LIN {X 0,Y 525.792,Z 279.61,A -85,B 0,C 180,E1 -4784.971,E2 -4784.971} C_VEL
LIN {X 0,Y 524.291,Z 269.507,A -85,B 0,C 180,E1 -4785.168,E2 -4785.168} C_VEL
LIN {X 0,Y 524.691,Z 248.989,A -85,B 0,C 180,E1 -4788.306,E2 -4788.306} C_VEL
LIN {X 0,Y 525.144,Z 230.381,A -85,B 0,C 180,E1 -4791.182,E2 -4791.182} C_VEL
LIN {X 0,Y 525.394,Z 217.304,A -85,B 0,C 180,E1 -4793.241,E2 -4793.241} C_VEL
LIN {X 0,Y 523.911,Z 209.225,A -85,B 0,C 180,E1 -4794.625,E2 -4794.625} C_VEL
LIN {X 0,Y 523.877,Z 209.232,A -85,B 0,C 180,E1 -4797.695,E2 -4797.695} C_VEL
LIN {X 0,Y 523.901,Z 209.222,A -85,B 0,C 180,E1 -4800.844,E2 -4800.844} C_VEL
LIN {X 0,Y 523.896,Z 209.229,A -85,B 0,C 180,E1 -4803.721,E2 -4803.721} C_VEL
LIN {X 0,Y 523.848,Z 209.228,A -85,B 0,C 180,E1 -4806.39,E2 -4806.39} C_VEL
LIN {X 0,Y 523.889,Z 209.223,A -85,B 0,C 180,E1 -4809.086,E2 -4809.086} C_VEL
LIN {X 0,Y 523.876,Z 209.227,A -85,B 0,C 180,E1 -4812.125,E2 -4812.125} C_VEL
LIN {X 0,Y 523.93,Z 209.22,A -85,B 0,C 180,E1 -4815.31,E2 -4815.31} C_VEL
LIN {X 0,Y 523.877,Z 209.223,A -85,B 0,C 180,E1 -4818.698,E2 -4818.698} C_VEL
LIN {X 0,Y 523.884,Z 209.224,A -85,B 0,C 180,E1 -4821.083,E2 -4821.083} C_VEL
LIN {X 0,Y 523.84,Z 209.235,A -85,B 0,C 180,E1 -4823.818,E2 -4823.818} C_VEL
LIN {X 0,Y 523.895,Z 209.221,A -85,B 0,C 180,E1 -4826.629,E2 -4826.629} C_VEL
LIN {X 0,Y 523.907,Z 209.224,A -85,B 0,C 180,E1 -4829.349,E2 -4829.349} C_VEL
LIN {X 0,Y 523.873,Z 209.225,A -85,B 0,C 180,E1 -4832.301,E2 -4832.301} C_VEL
LIN {X 0,Y 523.895,Z 209.227,A -85,B 0,C 180,E1 -4835.423,E2 -4835.423} C_VEL
LIN {X 0,Y 523.934,Z 209.221,A -85,B 0,C 180,E1 -4837.936,E2 -4837.936} C_VEL
LIN {X 0,Y 523.922,Z 209.218,A -85,B 0,C 180,E1 -4840.402,E2 -4840.402} C_VEL
LIN {X 0,Y 523.923,Z 209.218,A -85,B 0,C 180,E1 -4842.832,E2 -4842.832} C_VEL
LIN {X 0,Y 523.957,Z 209.217,A -85,B 0,C 180,E1 -4845.232,E2 -4845.232} C_VEL
LIN {X 0,Y 523.95,Z 209.214,A -85,B 0,C 180,E1 -4848.389,E2 -4848.389} C_VEL
LIN {X 0,Y 523.935,Z 209.225,A -85,B 0,C 180,E1 -4851.511,E2 -4851.511} C_VEL
LIN {X 0,Y 524.022,Z 209.205,A -85,B 0,C 180,E1 -4854.609,E2 -4854.609} C_VEL
LIN {X 0,Y 524.084,Z 209.204,A -85,B 0,C 180,E1 -4857.69,E2 -4857.69} C_VEL
LIN {X 0,Y 524.074,Z 209.201,A -85,B 0,C 180,E1 -4859.996,E2 -4859.996} C_VEL
LIN {X 0,Y 524.016,Z 209.209,A -85,B 0,C 180,E1 -4863.071,E2 -4863.071} C_VEL
LIN {X 0,Y 523.977,Z 209.212,A -85,B 0,C 180,E1 -4866.155,E2 -4866.155} C_VEL
LIN {X 0,Y 523.926,Z 209.223,A -85,B 0,C 180,E1 -4869.258,E2 -4869.258} C_VEL
LIN {X 0,Y 523.973,Z 209.216,A -85,B 0,C 180,E1 -4871.73,E2 -4871.73} C_VEL
LIN {X 0,Y 523.957,Z 209.217,A -85,B 0,C 180,E1 -4875.043,E2 -4875.043} C_VEL
LIN {X 0,Y 523.917,Z 209.22,A -85,B 0,C 180,E1 -4877.965,E2 -4877.965} C_VEL
LIN {X 0,Y 523.928,Z 209.217,A -85,B 0,C 180,E1 -4880.406,E2 -4880.406} C_VEL
LIN {X 0,Y 523.876,Z 209.226,A -85,B 0,C 180,E1 -4882.889,E2 -4882.889} C_VEL
LIN {X 0,Y 523.877,Z 209.232,A -85,B 0,C 180,E1 -4885.416,E2 -4885.416} C_VEL
LIN {X 0,Y 523.92,Z 209.219,A -85,B 0,C 180,E1 -4887.995,E2 -4887.995} C_VEL
LIN {X 0,Y 523.901,Z 209.223,A -85,B 0,C 180,E1 -4890.849,E2 -4890.849} C_VEL
LIN {X 0,Y 523.918,Z 209.222,A -85,B 0,C 180,E1 -4893.73,E2 -4893.73} C_VEL
LIN {X 0,Y 523.859,Z 209.225,A -85,B 0,C 180,E1 -4896.397,E2 -4896.397} C_VEL
LIN {X 0,Y 523.875,Z 209.229,A -85,B 0,C 180,E1 -4899.08,E2 -4899.08} C_VEL
LIN {X 0,Y 523.906,Z 209.22,A -85,B 0,C 180,E1 -4902.115,E2 -4902.115} C_VEL
LIN {X 0,Y 523.905,Z 209.229,A -85,B 0,C 180,E1 -4905.305,E2 -4905.305} C_VEL
LIN {X 0,Y 523.869,Z 209.227,A -85,B 0,C 180,E1 -4906.862,E2 -4906.862} C_VEL
LIN {X 0,Y 523.192,Z 209.315,A -85,B 0,C 180,E1 -4907.504,E2 -4907.504} C_VEL
LIN {X 0,Y 520.325,Z 209.666,A -85,B 0,C 180,E1 -4908.545,E2 -4908.545} C_VEL
LIN {X 0,Y 517.918,Z 209.973,A -85,B 0,C 180,E1 -4909.384,E2 -4909.384} C_VEL
LIN {X 0,Y 516.902,Z 210.093,A -85,B 0,C 180,E1 -4910.032,E2 -4910.032} C_VEL
LIN {X 0,Y 516.828,Z 210.101,A -85,B 0,C 180,E1 -4910.251,E2 -4910.251} C_VEL
LIN {X 0,Y 516.836,Z 210.108,A -85,B 0,C 180,E1 -4913.337,E2 -4913.337} C_VEL
LIN {X 0,Y 516.856,Z 210.098,A -85,B 0,C 180,E1 -4916.118,E2 -4916.118} C_VEL
LIN {X 0,Y 516.835,Z 210.105,A -85,B 0,C 180,E1 -4918.932,E2 -4918.932} C_VEL
LIN {X 0,Y 516.865,Z 210.1,A -85,B 0,C 180,E1 -4921.582,E2 -4921.582} C_VEL
LIN {X 0,Y 516.871,Z 210.096,A -85,B 0,C 180,E1 -4924.208,E2 -4924.208} C_VEL
LIN {X 0,Y 516.842,Z 210.103,A -85,B 0,C 180,E1 -4926.776,E2 -4926.776} C_VEL
LIN {X 0,Y 516.876,Z 210.097,A -85,B 0,C 180,E1 -4929.729,E2 -4929.729} C_VEL
LIN {X 0,Y 516.878,Z 210.097,A -85,B 0,C 180,E1 -4932.595,E2 -4932.595} C_VEL
LIN {X 0,Y 516.875,Z 210.103,A -85,B 0,C 180,E1 -4935.028,E2 -4935.028} C_VEL
LIN {X 0,Y 516.937,Z 210.088,A -85,B 0,C 180,E1 -4938.233,E2 -4938.233} C_VEL
LIN {X 0,Y 516.908,Z 210.096,A -85,B 0,C 180,E1 -4941.399,E2 -4941.399} C_VEL
LIN {X 0,Y 516.956,Z 210.086,A -85,B 0,C 180,E1 -4943.756,E2 -4943.756} C_VEL
LIN {X 0,Y 516.983,Z 210.089,A -85,B 0,C 180,E1 -4946.883,E2 -4946.883} C_VEL
LIN {X 0,Y 517.014,Z 210.078,A -85,B 0,C 180,E1 -4950,E2 -4950} C_VEL
LIN {X 0,Y 516.983,Z 210.09,A -85,B 0,C 180,E1 -4953.117,E2 -4953.117} C_VEL
LIN {X 0,Y 516.956,Z 210.086,A -85,B 0,C 180,E1 -4956.244,E2 -4956.244} C_VEL
LIN {X 0,Y 516.909,Z 210.096,A -85,B 0,C 180,E1 -4958.601,E2 -4958.601} C_VEL
LIN {X 0,Y 516.916,Z 210.095,A -85,B 0,C 180,E1 -4961.825,E2 -4961.825} C_VEL
LIN {X 0,Y 516.944,Z 210.255,A -85,B 0,C 180,E1 -4963.163,E2 -4963.163} C_VEL
LIN {X 0,Y 517.496,Z 216.237,A -85,B 0,C 180,E1 -4964.35,E2 -4964.35} C_VEL
LIN {X 0,Y 517.255,Z 231.009,A -85,B 0,C 180,E1 -4967.188,E2 -4967.188} C_VEL
LIN {X 0,Y 517.241,Z 233.79,A -85,B 0,C 180,E1 -4967.699,E2 -4967.699} C_VEL
LIN {X 0,Y 519.076,Z 243.862,A -85,B 0,C 180,E1 -4967.899,E2 -4967.899} C_VEL
LIN {X 0,Y 518.599,Z 340.175,A -85,B 0,C 180,E1 -4969.262,E2 -4969.262} C_VEL
LIN {X 0,Y 518.408,Z 353.794,A -85,B 0,C 180,E1 -4969.617,E2 -4969.617} C_VEL
LIN {X 0,Y 518.174,Z 366.867,A -85,B 0,C 180,E1 -4970.129,E2 -4970.129} C_VEL
LIN {X 0,Y 517.935,Z 378.637,A -85,B 0,C 180,E1 -4970.762,E2 -4970.762} C_VEL
LIN {X 0,Y 517.624,Z 389.477,A -85,B 0,C 180,E1 -4971.505,E2 -4971.505} C_VEL
LIN {X 0,Y 517.313,Z 399.511,A -85,B 0,C 180,E1 -4972.358,E2 -4972.358} C_VEL
LIN {X 0,Y 516.983,Z 409.671,A -85,B 0,C 180,E1 -4973.43,E2 -4973.43} C_VEL
LIN {X 0,Y 516.771,Z 418.579,A -85,B 0,C 180,E1 -4974.607,E2 -4974.607} C_VEL
LIN {X 0,Y 516.59,Z 425.889,A -85,B 0,C 180,E1 -4975.807,E2 -4975.807} C_VEL
LIN {X 0,Y 516.421,Z 432.17,A -85,B 0,C 180,E1 -4977.122,E2 -4977.122} C_VEL
LIN {X 0,Y 516.366,Z 437.002,A -85,B 0,C 180,E1 -4978.448,E2 -4978.448} C_VEL
LIN {X 0,Y 516.286,Z 439.701,A -85,B 0,C 180,E1 -4979.416,E2 -4979.416} C_VEL
LIN {X 0,Y 516.188,Z 442.581,A -85,B 0,C 180,E1 -4980.949,E2 -4980.949} C_VEL
LIN {X 0,Y 516.18,Z 443.91,A -85,B 0,C 180,E1 -4982.432,E2 -4982.432} C_VEL
LIN {X 0,Y 516.185,Z 443.757,A -85,B 0,C 180,E1 -4983.932,E2 -4983.932} C_VEL
LIN {X 0,Y 516.157,Z 442.467,A -85,B 0,C 180,E1 -4985.231,E2 -4985.231} C_VEL
LIN {X 0,Y 516.309,Z 439.445,A -85,B 0,C 180,E1 -4986.792,E2 -4986.792} C_VEL
LIN {X 0,Y 516.375,Z 434.854,A -85,B 0,C 180,E1 -4988.29,E2 -4988.29} C_VEL
LIN {X 0,Y 516.512,Z 430.235,A -85,B 0,C 180,E1 -4989.417,E2 -4989.417} C_VEL
LIN {X 0,Y 516.652,Z 423.229,A -85,B 0,C 180,E1 -4990.762,E2 -4990.762} C_VEL
LIN {X 0,Y 516.809,Z 416.576,A -85,B 0,C 180,E1 -4991.784,E2 -4991.784} C_VEL
LIN {X 0,Y 517.114,Z 408.481,A -85,B 0,C 180,E1 -4992.806,E2 -4992.806} C_VEL
LIN {X 0,Y 517.385,Z 398.328,A -85,B 0,C 180,E1 -4993.848,E2 -4993.848} C_VEL
LIN {X 0,Y 517.639,Z 388.752,A -85,B 0,C 180,E1 -4994.647,E2 -4994.647} C_VEL
LIN {X 0,Y 517.952,Z 377.818,A -85,B 0,C 180,E1 -4995.385,E2 -4995.385} C_VEL
LIN {X 0,Y 518.222,Z 365.8,A -85,B 0,C 180,E1 -4996.011,E2 -4996.011} C_VEL
LIN {X 0,Y 518.452,Z 352.312,A -85,B 0,C 180,E1 -4996.523,E2 -4996.523} C_VEL
LIN {X 0,Y 518.625,Z 339.718,A -85,B 0,C 180,E1 -4996.837,E2 -4996.837} C_VEL
LIN {X 0,Y 518.974,Z 242.983,A -85,B 0,C 180,E1 -4998.209,E2 -4998.209} C_VEL
LIN {X 0,Y 517.231,Z 233.482,A -85,B 0,C 180,E1 -4998.412,E2 -4998.412} C_VEL
LIN {X 0,Y 517.389,Z 217.337,A -85,B 0,C 180,E1 -5001.338,E2 -5001.338} C_VEL
LIN {X 0,Y 517.232,Z 211.916,A -85,B 0,C 180,E1 -5002.314,E2 -5002.314} C_VEL
LIN {X 0,Y 516.926,Z 210.098,A -85,B 0,C 180,E1 -5002.656,E2 -5002.656} C_VEL
LIN {X 0,Y 516.878,Z 210.098,A -85,B 0,C 180,E1 -5006.037,E2 -5006.037} C_VEL
LIN {X 0,Y 516.856,Z 210.107,A -85,B 0,C 180,E1 -5008.94,E2 -5008.94} C_VEL
LIN {X 0,Y 516.89,Z 210.097,A -85,B 0,C 180,E1 -5011.59,E2 -5011.59} C_VEL
LIN {X 0,Y 516.9,Z 210.093,A -85,B 0,C 180,E1 -5014.216,E2 -5014.216} C_VEL
LIN {X 0,Y 516.841,Z 210.107,A -85,B 0,C 180,E1 -5016.781,E2 -5016.781} C_VEL
LIN {X 0,Y 516.911,Z 210.093,A -85,B 0,C 180,E1 -5019.736,E2 -5019.736} C_VEL
LIN {X 0,Y 516.902,Z 210.098,A -85,B 0,C 180,E1 -5022.601,E2 -5022.601} C_VEL
LIN {X 0,Y 516.917,Z 210.097,A -85,B 0,C 180,E1 -5025.035,E2 -5025.035} C_VEL
LIN {X 0,Y 516.983,Z 210.084,A -85,B 0,C 180,E1 -5028.239,E2 -5028.239} C_VEL
LIN {X 0,Y 516.939,Z 210.089,A -85,B 0,C 180,E1 -5031.404,E2 -5031.404} C_VEL
LIN {X 0,Y 516.979,Z 210.083,A -85,B 0,C 180,E1 -5033.761,E2 -5033.761} C_VEL
LIN {X 0,Y 516.995,Z 210.088,A -85,B 0,C 180,E1 -5036.888,E2 -5036.888} C_VEL
LIN {X 0,Y 517.065,Z 210.073,A -85,B 0,C 180,E1 -5040.004,E2 -5040.004} C_VEL
LIN {X 0,Y 517.062,Z 210.074,A -85,B 0,C 180,E1 -5042.341,E2 -5042.341} C_VEL
LIN {X 0,Y 517.005,Z 210.078,A -85,B 0,C 180,E1 -5045.464,E2 -5045.464} C_VEL
LIN {X 0,Y 516.944,Z 210.087,A -85,B 0,C 180,E1 -5047.818,E2 -5047.818} C_VEL
LIN {X 0,Y 516.935,Z 210.093,A -85,B 0,C 180,E1 -5050.976,E2 -5050.976} C_VEL
LIN {X 0,Y 516.88,Z 210.097,A -85,B 0,C 180,E1 -5054.17,E2 -5054.17} C_VEL
LIN {X 0,Y 516.896,Z 210.102,A -85,B 0,C 180,E1 -5056.594,E2 -5056.594} C_VEL
LIN {X 0,Y 516.888,Z 210.096,A -85,B 0,C 180,E1 -5059.049,E2 -5059.049} C_VEL
LIN {X 0,Y 516.882,Z 210.094,A -85,B 0,C 180,E1 -5061.541,E2 -5061.541} C_VEL
LIN {X 0,Y 516.856,Z 210.104,A -85,B 0,C 180,E1 -5064.354,E2 -5064.354} C_VEL
LIN {X 0,Y 516.874,Z 210.095,A -85,B 0,C 180,E1 -5067.539,E2 -5067.539} C_VEL
LIN {X 0,Y 516.856,Z 210.102,A -85,B 0,C 180,E1 -5070.209,E2 -5070.209} C_VEL
LIN {X 0,Y 516.88,Z 210.096,A -85,B 0,C 180,E1 -5072.951,E2 -5072.951} C_VEL
LIN {X 0,Y 516.816,Z 210.105,A -85,B 0,C 180,E1 -5075.788,E2 -5075.788} C_VEL
LIN {X 0,Y 516.863,Z 210.102,A -85,B 0,C 180,E1 -5078.72,E2 -5078.72} C_VEL
LIN {X 0,Y 516.84,Z 210.103,A -85,B 0,C 180,E1 -5081.785,E2 -5081.785} C_VEL
LIN {X 0,Y 516.901,Z 210.095,A -85,B 0,C 180,E1 -5085.009,E2 -5085.009} C_VEL
LIN {X 0,Y 516.832,Z 210.11,A -85,B 0,C 180,E1 -5088.412,E2 -5088.412} C_VEL
LIN {X 0,Y 516.855,Z 210.099,A -85,B 0,C 180,E1 -5091.283,E2 -5091.283} C_VEL
LIN {X 0,Y 516.831,Z 210.106,A -85,B 0,C 180,E1 -5094.679,E2 -5094.679} C_VEL
LIN {X 0,Y 516.869,Z 210.1,A -85,B 0,C 180,E1 -5097.464,E2 -5097.464} C_VEL
LIN {X 0,Y 516.845,Z 210.108,A -85,B 0,C 180,E1 -5100.492,E2 -5100.492} C_VEL
LIN {X 0,Y 516.818,Z 210.106,A -85,B 0,C 180,E1 -5103.337,E2 -5103.337} C_VEL
LIN {X 0,Y 516.899,Z 210.289,A -85,B 0,C 180,E1 -5105.44,E2 -5105.44} C_VEL
LIN {X 0,Y 518.322,Z 218.758,A -85,B 0,C 180,E1 -5106.846,E2 -5106.846} C_VEL
LIN {X 0,Y 517.95,Z 236.058,A -85,B 0,C 180,E1 -5109.549,E2 -5109.549} C_VEL
LIN {X 0,Y 517.547,Z 254.75,A -85,B 0,C 180,E1 -5112.438,E2 -5112.438} C_VEL
LIN {X 0,Y 517.227,Z 269.021,A -85,B 0,C 180,E1 -5114.622,E2 -5114.622} C_VEL
LIN {X 0,Y 519.018,Z 281.084,A -85,B 0,C 180,E1 -5114.856,E2 -5114.856} C_VEL
LIN {X 0,Y 518.579,Z 377.987,A -85,B 0,C 180,E1 -5116.231,E2 -5116.231} C_VEL
LIN {X 0,Y 518.314,Z 391.113,A -85,B 0,C 180,E1 -5116.574,E2 -5116.574} C_VEL
LIN {X 0,Y 518.039,Z 403.784,A -85,B 0,C 180,E1 -5117.065,E2 -5117.065} C_VEL
LIN {X 0,Y 517.789,Z 415.585,A -85,B 0,C 180,E1 -5117.69,E2 -5117.69} C_VEL
LIN {X 0,Y 517.501,Z 426.729,A -85,B 0,C 180,E1 -5118.445,E2 -5118.445} C_VEL
LIN {X 0,Y 517.219,Z 437.236,A -85,B 0,C 180,E1 -5119.331,E2 -5119.331} C_VEL
LIN {X 0,Y 516.924,Z 445.825,A -85,B 0,C 180,E1 -5120.216,E2 -5120.216} C_VEL
LIN {X 0,Y 516.705,Z 453.75,A -85,B 0,C 180,E1 -5121.198,E2 -5121.198} C_VEL
LIN {X 0,Y 516.529,Z 461.492,A -85,B 0,C 180,E1 -5122.377,E2 -5122.377} C_VEL
LIN {X 0,Y 516.385,Z 468.624,A -85,B 0,C 180,E1 -5123.749,E2 -5123.749} C_VEL
LIN {X 0,Y 516.313,Z 473.37,A -85,B 0,C 180,E1 -5124.924,E2 -5124.924} C_VEL
LIN {X 0,Y 516.354,Z 477,A -85,B 0,C 180,E1 -5126.098,E2 -5126.098} C_VEL
LIN {X 0,Y 516.284,Z 478.87,A -85,B 0,C 180,E1 -5126.879,E2 -5126.879} C_VEL
LIN {X 0,Y 516.263,Z 480.273,A -85,B 0,C 180,E1 -5127.66,E2 -5127.66} C_VEL
LIN {X 0,Y 516.164,Z 481.885,A -85,B 0,C 180,E1 -5129.22,E2 -5129.22} C_VEL
LIN {X 0,Y 516.161,Z 482.105,A -85,B 0,C 180,E1 -5130,E2 -5130} C_VEL
LIN {X 0,Y 516.193,Z 481.283,A -85,B 0,C 180,E1 -5131.56,E2 -5131.56} C_VEL
LIN {X 0,Y 516.263,Z 480.29,A -85,B 0,C 180,E1 -5132.341,E2 -5132.341} C_VEL
LIN {X 0,Y 516.284,Z 478.892,A -85,B 0,C 180,E1 -5133.121,E2 -5133.121} C_VEL
LIN {X 0,Y 516.312,Z 475.95,A -85,B 0,C 180,E1 -5134.293,E2 -5134.293} C_VEL
LIN {X 0,Y 516.369,Z 471.966,A -85,B 0,C 180,E1 -5135.467,E2 -5135.467} C_VEL
LIN {X 0,Y 516.394,Z 466.783,A -85,B 0,C 180,E1 -5136.654,E2 -5136.654} C_VEL
LIN {X 0,Y 516.546,Z 460.374,A -85,B 0,C 180,E1 -5137.82,E2 -5137.82} C_VEL
LIN {X 0,Y 516.758,Z 452.318,A -85,B 0,C 180,E1 -5138.998,E2 -5138.998} C_VEL
LIN {X 0,Y 516.95,Z 444.106,A -85,B 0,C 180,E1 -5139.982,E2 -5139.982} C_VEL
LIN {X 0,Y 517.288,Z 434.094,A -85,B 0,C 180,E1 -5140.965,E2 -5140.965} C_VEL
LIN {X 0,Y 517.569,Z 424.203,A -85,B 0,C 180,E1 -5141.752,E2 -5141.752} C_VEL
LIN {X 0,Y 517.851,Z 413.036,A -85,B 0,C 180,E1 -5142.465,E2 -5142.465} C_VEL
LIN {X 0,Y 518.115,Z 400.511,A -85,B 0,C 180,E1 -5143.082,E2 -5143.082} C_VEL
LIN {X 0,Y 518.395,Z 388.177,A -85,B 0,C 180,E1 -5143.524,E2 -5143.524} C_VEL
LIN {X 0,Y 518.626,Z 375.486,A -85,B 0,C 180,E1 -5143.818,E2 -5143.818} C_VEL
LIN {X 0,Y 518.866,Z 279.935,A -85,B 0,C 180,E1 -5145.168,E2 -5145.168} C_VEL
LIN {X 0,Y 517.279,Z 269.248,A -85,B 0,C 180,E1 -5145.38,E2 -5145.38} C_VEL
LIN {X 0,Y 517.743,Z 248.473,A -85,B 0,C 180,E1 -5148.602,E2 -5148.602} C_VEL
LIN {X 0,Y 518.21,Z 230.161,A -85,B 0,C 180,E1 -5151.479,E2 -5151.479} C_VEL
LIN {X 0,Y 518.434,Z 218.384,A -85,B 0,C 180,E1 -5153.36,E2 -5153.36} C_VEL
LIN {X 0,Y 516.888,Z 210.1,A -85,B 0,C 180,E1 -5154.78,E2 -5154.78} C_VEL
LIN {X 0,Y 516.826,Z 210.11,A -85,B 0,C 180,E1 -5157.881,E2 -5157.881} C_VEL
LIN {X 0,Y 516.842,Z 210.105,A -85,B 0,C 180,E1 -5160.206,E2 -5160.206} C_VEL
LIN {X 0,Y 516.818,Z 210.103,A -85,B 0,C 180,E1 -5162.952,E2 -5162.952} C_VEL
LIN {X 0,Y 516.8,Z 210.114,A -85,B 0,C 180,E1 -5165.785,E2 -5165.785} C_VEL
LIN {X 0,Y 516.853,Z 210.098,A -85,B 0,C 180,E1 -5168.717,E2 -5168.717} C_VEL
LIN {X 0,Y 516.827,Z 210.111,A -85,B 0,C 180,E1 -5171.782,E2 -5171.782} C_VEL
LIN {X 0,Y 516.867,Z 210.097,A -85,B 0,C 180,E1 -5175.001,E2 -5175.001} C_VEL
LIN {X 0,Y 516.832,Z 210.103,A -85,B 0,C 180,E1 -5178.214,E2 -5178.214} C_VEL
LIN {X 0,Y 516.848,Z 210.102,A -85,B 0,C 180,E1 -5181.278,E2 -5181.278} C_VEL
LIN {X 0,Y 516.822,Z 210.102,A -85,B 0,C 180,E1 -5184.675,E2 -5184.675} C_VEL
LIN {X 0,Y 516.864,Z 210.103,A -85,B 0,C 180,E1 -5187.46,E2 -5187.46} C_VEL
LIN {X 0,Y 516.839,Z 210.1,A -85,B 0,C 180,E1 -5190.488,E2 -5190.488} C_VEL
LIN {X 0,Y 516.818,Z 210.107,A -85,B 0,C 180,E1 -5193.333,E2 -5193.333} C_VEL
LIN {X 0,Y 516.868,Z 210.101,A -85,B 0,C 180,E1 -5195.923,E2 -5195.923} C_VEL
LIN {X 0,Y 516.859,Z 210.098,A -85,B 0,C 180,E1 -5198.458,E2 -5198.458} C_VEL
LIN {X 0,Y 516.86,Z 210.098,A -85,B 0,C 180,E1 -5200.95,E2 -5200.95} C_VEL
LIN {X 0,Y 516.867,Z 210.103,A -85,B 0,C 180,E1 -5203.405,E2 -5203.405} C_VEL
LIN {X 0,Y 516.865,Z 210.102,A -85,B 0,C 180,E1 -5205.829,E2 -5205.829} C_VEL
LIN {X 0,Y 516.914,Z 210.092,A -85,B 0,C 180,E1 -5208.229,E2 -5208.229} C_VEL
LIN {X 0,Y 516.908,Z 210.098,A -85,B 0,C 180,E1 -5211.395,E2 -5211.395} C_VEL
LIN {X 0,Y 516.973,Z 210.083,A -85,B 0,C 180,E1 -5214.535,E2 -5214.535} C_VEL
LIN {X 0,Y 517.055,Z 210.08,A -85,B 0,C 180,E1 -5217.659,E2 -5217.659} C_VEL
LIN {X 0,Y 517.044,Z 210.077,A -85,B 0,C 180,E1 -5219.996,E2 -5219.996} C_VEL
LIN {X 0,Y 517.055,Z 210.073,A -85,B 0,C 180,E1 -5222.332,E2 -5222.332} C_VEL
LIN {X 0,Y 516.961,Z 210.094,A -85,B 0,C 180,E1 -5225.456,E2 -5225.456} C_VEL
LIN {X 0,Y 516.907,Z 210.092,A -85,B 0,C 180,E1 -5228.596,E2 -5228.596} C_VEL
LIN {X 0,Y 516.931,Z 210.092,A -85,B 0,C 180,E1 -5231.802,E2 -5231.802} C_VEL
LIN {X 0,Y 516.91,Z 210.096,A -85,B 0,C 180,E1 -5235.137,E2 -5235.137} C_VEL
LIN {X 0,Y 516.885,Z 210.095,A -85,B 0,C 180,E1 -5238.218,E2 -5238.218} C_VEL
LIN {X 0,Y 516.875,Z 210.096,A -85,B 0,C 180,E1 -5240.697,E2 -5240.697} C_VEL
LIN {X 0,Y 516.852,Z 210.099,A -85,B 0,C 180,E1 -5244.069,E2 -5244.069} C_VEL
LIN {X 0,Y 516.871,Z 210.097,A -85,B 0,C 180,E1 -5246.654,E2 -5246.654} C_VEL
LIN {X 0,Y 516.871,Z 210.103,A -85,B 0,C 180,E1 -5249.518,E2 -5249.518} C_VEL
LIN {X 0,Y 516.856,Z 210.098,A -85,B 0,C 180,E1 -5252.539,E2 -5252.539} C_VEL
LIN {X 0,Y 516.824,Z 210.111,A -85,B 0,C 180,E1 -5255.325,E2 -5255.325} C_VEL
LIN {X 0,Y 516.835,Z 210.102,A -85,B 0,C 180,E1 -5257.938,E2 -5257.938} C_VEL
LIN {X 0,Y 516.838,Z 210.102,A -85,B 0,C 180,E1 -5260.737,E2 -5260.737} C_VEL
LIN {X 0,Y 516.837,Z 210.103,A -85,B 0,C 180,E1 -5262.827,E2 -5262.827} C_VEL
LIN {X 0,Y 516.873,Z 210.101,A -85,B 0,C 180,E1 -5265.006,E2 -5265.006} C_VEL
LIN {X 0,Y 516.87,Z 210.096,A -85,B 0,C 180,E1 -5268.394,E2 -5268.394} C_VEL
LIN {X 0,Y 516.828,Z 210.101,A -85,B 0,C 180,E1 -5270.251,E2 -5270.251} C_VEL
LIN {X 0,Y 516.188,Z 210.187,A -85,B 0,C 180,E1 -5270.901,E2 -5270.901} C_VEL
LIN {X 0,Y 513.348,Z 210.542,A -85,B 0,C 180,E1 -5271.957,E2 -5271.957} C_VEL
LIN {X 0,Y 510.926,Z 210.844,A -85,B 0,C 180,E1 -5272.807,E2 -5272.807} C_VEL
LIN {X 0,Y 509.874,Z 210.974,A -85,B 0,C 180,E1 -5273.463,E2 -5273.463} C_VEL
LIN {X 0,Y 509.784,Z 210.982,A -85,B 0,C 180,E1 -5273.686,E2 -5273.686} C_VEL
LIN {X 0,Y 509.805,Z 210.977,A -85,B 0,C 180,E1 -5276.536,E2 -5276.536} C_VEL
LIN {X 0,Y 509.792,Z 210.985,A -85,B 0,C 180,E1 -5279.332,E2 -5279.332} C_VEL
LIN {X 0,Y 509.836,Z 210.972,A -85,B 0,C 180,E1 -5282.052,E2 -5282.052} C_VEL
LIN {X 0,Y 509.821,Z 210.977,A -85,B 0,C 180,E1 -5284.702,E2 -5284.702} C_VEL
LIN {X 0,Y 509.821,Z 210.979,A -85,B 0,C 180,E1 -5287.44,E2 -5287.44} C_VEL
LIN {X 0,Y 509.854,Z 210.971,A -85,B 0,C 180,E1 -5289.843,E2 -5289.843} C_VEL
LIN {X 0,Y 509.843,Z 210.972,A -85,B 0,C 180,E1 -5292.347,E2 -5292.347} C_VEL
LIN {X 0,Y 509.8,Z 210.979,A -85,B 0,C 180,E1 -5295.633,E2 -5295.633} C_VEL
LIN {X 0,Y 509.87,Z 210.974,A -85,B 0,C 180,E1 -5298.874,E2 -5298.874} C_VEL
LIN {X 0,Y 509.904,Z 210.964,A -85,B 0,C 180,E1 -5302.078,E2 -5302.078} C_VEL
LIN {X 0,Y 509.948,Z 210.96,A -85,B 0,C 180,E1 -5304.464,E2 -5304.464} C_VEL
LIN {X 0,Y 509.99,Z 210.955,A -85,B 0,C 180,E1 -5307.631,E2 -5307.631} C_VEL
LIN {X 0,Y 509.985,Z 210.954,A -85,B 0,C 180,E1 -5310,E2 -5310} C_VEL
LIN {X 0,Y 509.924,Z 210.968,A -85,B 0,C 180,E1 -5313.16,E2 -5313.16} C_VEL
LIN {X 0,Y 509.927,Z 210.962,A -85,B 0,C 180,E1 -5316.33,E2 -5316.33} C_VEL
LIN {X 0,Y 509.884,Z 210.973,A -85,B 0,C 180,E1 -5318.72,E2 -5318.72} C_VEL
LIN {X 0,Y 509.885,Z 210.971,A -85,B 0,C 180,E1 -5321.932,E2 -5321.932} C_VEL
LIN {X 0,Y 509.89,Z 211.067,A -85,B 0,C 180,E1 -5323.018,E2 -5323.018} C_VEL
LIN {X 0,Y 510.539,Z 217.685,A -85,B 0,C 180,E1 -5324.346,E2 -5324.346} C_VEL
LIN {X 0,Y 510.238,Z 232.559,A -85,B 0,C 180,E1 -5327.225,E2 -5327.225} C_VEL
LIN {X 0,Y 510.261,Z 233.996,A -85,B 0,C 180,E1 -5327.483,E2 -5327.483} C_VEL
LIN {X 0,Y 512.257,Z 245.073,A -85,B 0,C 180,E1 -5327.706,E2 -5327.706} C_VEL
LIN {X 0,Y 511.722,Z 340.827,A -85,B 0,C 180,E1 -5329.085,E2 -5329.085} C_VEL
LIN {X 0,Y 511.511,Z 354.047,A -85,B 0,C 180,E1 -5329.436,E2 -5329.436} C_VEL
LIN {X 0,Y 511.277,Z 366.832,A -85,B 0,C 180,E1 -5329.942,E2 -5329.942} C_VEL
LIN {X 0,Y 510.998,Z 379.302,A -85,B 0,C 180,E1 -5330.622,E2 -5330.622} C_VEL
LIN {X 0,Y 510.644,Z 390.267,A -85,B 0,C 180,E1 -5331.39,E2 -5331.39} C_VEL
LIN {X 0,Y 510.298,Z 401.247,A -85,B 0,C 180,E1 -5332.355,E2 -5332.355} C_VEL
LIN {X 0,Y 509.972,Z 410.265,A -85,B 0,C 180,E1 -5333.341,E2 -5333.341} C_VEL
LIN {X 0,Y 509.748,Z 419.017,A -85,B 0,C 180,E1 -5334.519,E2 -5334.519} C_VEL
LIN {X 0,Y 509.525,Z 426.382,A -85,B 0,C 180,E1 -5335.752,E2 -5335.752} C_VEL
LIN {X 0,Y 509.354,Z 432.603,A -85,B 0,C 180,E1 -5337.085,E2 -5337.085} C_VEL
LIN {X 0,Y 509.301,Z 437.395,A -85,B 0,C 180,E1 -5338.428,E2 -5338.428} C_VEL
LIN {X 0,Y 509.16,Z 440.923,A -85,B 0,C 180,E1 -5339.795,E2 -5339.795} C_VEL
LIN {X 0,Y 509.094,Z 443.162,A -85,B 0,C 180,E1 -5341.155,E2 -5341.155} C_VEL
LIN {X 0,Y 509.077,Z 444.22,A -85,B 0,C 180,E1 -5342.648,E2 -5342.648} C_VEL
LIN {X 0,Y 509.082,Z 443.935,A -85,B 0,C 180,E1 -5344.087,E2 -5344.087} C_VEL
LIN {X 0,Y 509.104,Z 442.425,A -85,B 0,C 180,E1 -5345.477,E2 -5345.477} C_VEL
LIN {X 0,Y 509.243,Z 439.719,A -85,B 0,C 180,E1 -5346.839,E2 -5346.839} C_VEL
LIN {X 0,Y 509.29,Z 435.891,A -85,B 0,C 180,E1 -5348.145,E2 -5348.145} C_VEL
LIN {X 0,Y 509.432,Z 430.849,A -85,B 0,C 180,E1 -5349.427,E2 -5349.427} C_VEL
LIN {X 0,Y 509.613,Z 423.769,A -85,B 0,C 180,E1 -5350.819,E2 -5350.819} C_VEL
LIN {X 0,Y 509.782,Z 416.879,A -85,B 0,C 180,E1 -5351.898,E2 -5351.898} C_VEL
LIN {X 0,Y 510.106,Z 408.598,A -85,B 0,C 180,E1 -5352.956,E2 -5352.956} C_VEL
LIN {X 0,Y 510.379,Z 399.397,A -85,B 0,C 180,E1 -5353.92,E2 -5353.92} C_VEL
LIN {X 0,Y 510.688,Z 388.417,A -85,B 0,C 180,E1 -5354.852,E2 -5354.852} C_VEL
LIN {X 0,Y 511.027,Z 378.028,A -85,B 0,C 180,E1 -5355.555,E2 -5355.555} C_VEL
LIN {X 0,Y 511.302,Z 366.059,A -85,B 0,C 180,E1 -5356.187,E2 -5356.187} C_VEL
LIN {X 0,Y 511.553,Z 352.701,A -85,B 0,C 180,E1 -5356.702,E2 -5356.702} C_VEL
LIN {X 0,Y 511.738,Z 339.562,A -85,B 0,C 180,E1 -5357.031,E2 -5357.031} C_VEL
LIN {X 0,Y 512.198,Z 244.126,A -85,B 0,C 180,E1 -5358.402,E2 -5358.402} C_VEL
LIN {X 0,Y 510.232,Z 233.768,A -85,B 0,C 180,E1 -5358.621,E2 -5358.621} C_VEL
LIN {X 0,Y 510.416,Z 218.102,A -85,B 0,C 180,E1 -5361.469,E2 -5361.469} C_VEL
LIN {X 0,Y 510.179,Z 212.733,A -85,B 0,C 180,E1 -5362.45,E2 -5362.45} C_VEL
LIN {X 0,Y 509.871,Z 210.977,A -85,B 0,C 180,E1 -5362.792,E2 -5362.792} C_VEL
LIN {X 0,Y 509.825,Z 210.978,A -85,B 0,C 180,E1 -5365.8,E2 -5365.8} C_VEL
LIN {X 0,Y 509.811,Z 210.983,A -85,B 0,C 180,E1 -5368.724,E2 -5368.724} C_VEL
LIN {X 0,Y 509.85,Z 210.979,A -85,B 0,C 180,E1 -5371.161,E2 -5371.161} C_VEL
LIN {X 0,Y 509.877,Z 210.968,A -85,B 0,C 180,E1 -5373.834,E2 -5373.834} C_VEL
LIN {X 0,Y 509.805,Z 210.979,A -85,B 0,C 180,E1 -5376.442,E2 -5376.442} C_VEL
LIN {X 0,Y 509.888,Z 210.967,A -85,B 0,C 180,E1 -5379.85,E2 -5379.85} C_VEL
LIN {X 0,Y 509.858,Z 210.977,A -85,B 0,C 180,E1 -5383.18,E2 -5383.18} C_VEL
LIN {X 0,Y 509.839,Z 210.973,A -85,B 0,C 180,E1 -5385.639,E2 -5385.639} C_VEL
LIN {X 0,Y 509.909,Z 210.971,A -85,B 0,C 180,E1 -5388.88,E2 -5388.88} C_VEL
LIN {X 0,Y 509.903,Z 210.964,A -85,B 0,C 180,E1 -5392.083,E2 -5392.083} C_VEL
LIN {X 0,Y 509.956,Z 210.962,A -85,B 0,C 180,E1 -5394.469,E2 -5394.469} C_VEL
LIN {X 0,Y 510.034,Z 210.947,A -85,B 0,C 180,E1 -5397.635,E2 -5397.635} C_VEL
LIN {X 0,Y 510.051,Z 210.953,A -85,B 0,C 180,E1 -5400.794,E2 -5400.794} C_VEL
LIN {X 0,Y 509.904,Z 210.967,A -85,B 0,C 180,E1 -5403.165,E2 -5403.165} C_VEL
LIN {X 0,Y 509.928,Z 210.963,A -85,B 0,C 180,E1 -5406.334,E2 -5406.334} C_VEL
LIN {X 0,Y 509.875,Z 210.974,A -85,B 0,C 180,E1 -5408.725,E2 -5408.725} C_VEL
LIN {X 0,Y 509.898,Z 210.966,A -85,B 0,C 180,E1 -5411.936,E2 -5411.936} C_VEL
LIN {X 0,Y 509.891,Z 210.967,A -85,B 0,C 180,E1 -5415.246,E2 -5415.246} C_VEL
LIN {X 0,Y 509.853,Z 210.976,A -85,B 0,C 180,E1 -5418.488,E2 -5418.488} C_VEL
LIN {X 0,Y 509.847,Z 210.974,A -85,B 0,C 180,E1 -5421.005,E2 -5421.005} C_VEL
LIN {X 0,Y 509.81,Z 210.975,A -85,B 0,C 180,E1 -5423.568,E2 -5423.568} C_VEL
LIN {X 0,Y 509.799,Z 210.983,A -85,B 0,C 180,E1 -5426.356,E2 -5426.356} C_VEL
LIN {X 0,Y 509.849,Z 210.974,A -85,B 0,C 180,E1 -5428.849,E2 -5428.849} C_VEL
LIN {X 0,Y 509.811,Z 210.976,A -85,B 0,C 180,E1 -5431.594,E2 -5431.594} C_VEL
LIN {X 0,Y 509.834,Z 210.98,A -85,B 0,C 180,E1 -5434.418,E2 -5434.418} C_VEL
LIN {X 0,Y 509.778,Z 210.98,A -85,B 0,C 180,E1 -5437.347,E2 -5437.347} C_VEL
LIN {X 0,Y 509.794,Z 210.986,A -85,B 0,C 180,E1 -5440.389,E2 -5440.389} C_VEL
LIN {X 0,Y 509.796,Z 210.98,A -85,B 0,C 180,E1 -5443.577,E2 -5443.577} C_VEL
LIN {X 0,Y 509.795,Z 210.987,A -85,B 0,C 180,E1 -5446.427,E2 -5446.427} C_VEL
LIN {X 0,Y 509.79,Z 210.98,A -85,B 0,C 180,E1 -5449.614,E2 -5449.614} C_VEL
LIN {X 0,Y 509.763,Z 210.987,A -85,B 0,C 180,E1 -5452.656,E2 -5452.656} C_VEL
LIN {X 0,Y 509.834,Z 210.977,A -85,B 0,C 180,E1 -5455.804,E2 -5455.804} C_VEL
LIN {X 0,Y 509.821,Z 210.981,A -85,B 0,C 180,E1 -5458.728,E2 -5458.728} C_VEL
LIN {X 0,Y 509.798,Z 210.986,A -85,B 0,C 180,E1 -5462.05,E2 -5462.05} C_VEL
LIN {X 0,Y 509.827,Z 211.067,A -85,B 0,C 180,E1 -5465.256,E2 -5465.256} C_VEL
LIN {X 0,Y 511.403,Z 220.464,A -85,B 0,C 180,E1 -5466.84,E2 -5466.84} C_VEL
LIN {X 0,Y 510.95,Z 237.782,A -85,B 0,C 180,E1 -5469.577,E2 -5469.577} C_VEL
LIN {X 0,Y 510.539,Z 255.633,A -85,B 0,C 180,E1 -5472.372,E2 -5472.372} C_VEL
LIN {X 0,Y 510.234,Z 268.741,A -85,B 0,C 180,E1 -5474.407,E2 -5474.407} C_VEL
LIN {X 0,Y 512.173,Z 283.028,A -85,B 0,C 180,E1 -5474.68,E2 -5474.68} C_VEL
LIN {X 0,Y 511.693,Z 377.582,A -85,B 0,C 180,E1 -5476.042,E2 -5476.042} C_VEL
LIN {X 0,Y 511.411,Z 390.748,A -85,B 0,C 180,E1 -5476.389,E2 -5476.389} C_VEL
LIN {X 0,Y 511.107,Z 403.442,A -85,B 0,C 180,E1 -5476.887,E2 -5476.887} C_VEL
LIN {X 0,Y 510.837,Z 415.13,A -85,B 0,C 180,E1 -5477.511,E2 -5477.511} C_VEL
LIN {X 0,Y 510.509,Z 426.417,A -85,B 0,C 180,E1 -5478.285,E2 -5478.285} C_VEL
LIN {X 0,Y 510.216,Z 436.934,A -85,B 0,C 180,E1 -5479.183,E2 -5479.183} C_VEL
LIN {X 0,Y 509.868,Z 445.528,A -85,B 0,C 180,E1 -5480.079,E2 -5480.079} C_VEL
LIN {X 0,Y 509.658,Z 453.461,A -85,B 0,C 180,E1 -5481.076,E2 -5481.076} C_VEL
LIN {X 0,Y 509.46,Z 461.209,A -85,B 0,C 180,E1 -5482.27,E2 -5482.27} C_VEL
LIN {X 0,Y 509.315,Z 468.347,A -85,B 0,C 180,E1 -5483.662,E2 -5483.662} C_VEL
LIN {X 0,Y 509.243,Z 473.098,A -85,B 0,C 180,E1 -5484.854,E2 -5484.854} C_VEL
LIN {X 0,Y 509.247,Z 476.731,A -85,B 0,C 180,E1 -5486.043,E2 -5486.043} C_VEL
LIN {X 0,Y 509.203,Z 478.604,A -85,B 0,C 180,E1 -5486.835,E2 -5486.835} C_VEL
LIN {X 0,Y 509.192,Z 480.009,A -85,B 0,C 180,E1 -5487.627,E2 -5487.627} C_VEL
LIN {X 0,Y 509.077,Z 481.623,A -85,B 0,C 180,E1 -5489.209,E2 -5489.209} C_VEL
LIN {X 0,Y 509.072,Z 481.843,A -85,B 0,C 180,E1 -5490,E2 -5490} C_VEL
LIN {X 0,Y 509.114,Z 481.023,A -85,B 0,C 180,E1 -5491.582,E2 -5491.582} C_VEL
LIN {X 0,Y 509.192,Z 480.03,A -85,B 0,C 180,E1 -5492.373,E2 -5492.373} C_VEL
LIN {X 0,Y 509.203,Z 478.63,A -85,B 0,C 180,E1 -5493.165,E2 -5493.165} C_VEL
LIN {X 0,Y 509.204,Z 475.686,A -85,B 0,C 180,E1 -5494.353,E2 -5494.353} C_VEL
LIN {X 0,Y 509.285,Z 471.701,A -85,B 0,C 180,E1 -5495.543,E2 -5495.543} C_VEL
LIN {X 0,Y 509.335,Z 465.666,A -85,B 0,C 180,E1 -5496.915,E2 -5496.915} C_VEL
LIN {X 0,Y 509.547,Z 458.865,A -85,B 0,C 180,E1 -5498.127,E2 -5498.127} C_VEL
LIN {X 0,Y 509.741,Z 450.548,A -85,B 0,C 180,E1 -5499.323,E2 -5499.323} C_VEL
LIN {X 0,Y 509.976,Z 442.015,A -85,B 0,C 180,E1 -5500.32,E2 -5500.32} C_VEL
LIN {X 0,Y 510.364,Z 431.478,A -85,B 0,C 180,E1 -5501.316,E2 -5501.316} C_VEL
LIN {X 0,Y 510.651,Z 420.416,A -85,B 0,C 180,E1 -5502.16,E2 -5502.16} C_VEL
LIN {X 0,Y 510.994,Z 409.604,A -85,B 0,C 180,E1 -5502.813,E2 -5502.813} C_VEL
LIN {X 0,Y 511.233,Z 397.796,A -85,B 0,C 180,E1 -5503.363,E2 -5503.363} C_VEL
LIN {X 0,Y 511.56,Z 385.106,A -85,B 0,C 180,E1 -5503.784,E2 -5503.784} C_VEL
LIN {X 0,Y 511.759,Z 372.086,A -85,B 0,C 180,E1 -5504.058,E2 -5504.058} C_VEL
LIN {X 0,Y 512.016,Z 280.767,A -85,B 0,C 180,E1 -5505.36,E2 -5505.36} C_VEL
LIN {X 0,Y 510.256,Z 269.037,A -85,B 0,C 180,E1 -5505.591,E2 -5505.591} C_VEL
LIN {X 0,Y 510.747,Z 249.527,A -85,B 0,C 180,E1 -5508.658,E2 -5508.658} C_VEL
LIN {X 0,Y 511.259,Z 231.235,A -85,B 0,C 180,E1 -5511.574,E2 -5511.574} C_VEL
LIN {X 0,Y 511.449,Z 219.463,A -85,B 0,C 180,E1 -5513.484,E2 -5513.484} C_VEL
LIN {X 0,Y 509.809,Z 210.982,A -85,B 0,C 180,E1 -5514.977,E2 -5514.977} C_VEL
LIN {X 0,Y 509.786,Z 210.986,A -85,B 0,C 180,E1 -5518.074,E2 -5518.074} C_VEL
LIN {X 0,Y 509.817,Z 210.978,A -85,B 0,C 180,E1 -5521.271,E2 -5521.271} C_VEL
LIN {X 0,Y 509.819,Z 210.976,A -85,B 0,C 180,E1 -5524.415,E2 -5524.415} C_VEL
LIN {X 0,Y 509.756,Z 210.985,A -85,B 0,C 180,E1 -5527.345,E2 -5527.345} C_VEL
LIN {X 0,Y 509.79,Z 210.979,A -85,B 0,C 180,E1 -5530.386,E2 -5530.386} C_VEL
LIN {X 0,Y 509.773,Z 210.987,A -85,B 0,C 180,E1 -5533.575,E2 -5533.575} C_VEL
LIN {X 0,Y 509.795,Z 210.978,A -85,B 0,C 180,E1 -5536.423,E2 -5536.423} C_VEL
LIN {X 0,Y 509.788,Z 210.986,A -85,B 0,C 180,E1 -5539.61,E2 -5539.61} C_VEL
LIN {X 0,Y 509.748,Z 210.983,A -85,B 0,C 180,E1 -5542.65,E2 -5542.65} C_VEL
LIN {X 0,Y 509.827,Z 210.981,A -85,B 0,C 180,E1 -5545.8,E2 -5545.8} C_VEL
LIN {X 0,Y 509.816,Z 210.975,A -85,B 0,C 180,E1 -5548.723,E2 -5548.723} C_VEL
LIN {X 0,Y 509.793,Z 210.981,A -85,B 0,C 180,E1 -5552.045,E2 -5552.045} C_VEL
LIN {X 0,Y 509.784,Z 210.979,A -85,B 0,C 180,E1 -5554.696,E2 -5554.696} C_VEL
LIN {X 0,Y 509.824,Z 210.98,A -85,B 0,C 180,E1 -5557.455,E2 -5557.455} C_VEL
LIN {X 0,Y 509.821,Z 210.974,A -85,B 0,C 180,E1 -5560.676,E2 -5560.676} C_VEL
LIN {X 0,Y 509.814,Z 210.978,A -85,B 0,C 180,E1 -5563.169,E2 -5563.169} C_VEL
LIN {X 0,Y 509.839,Z 210.981,A -85,B 0,C 180,E1 -5565.63,E2 -5565.63} C_VEL
LIN {X 0,Y 509.848,Z 210.972,A -85,B 0,C 180,E1 -5568.869,E2 -5568.869} C_VEL
LIN {X 0,Y 509.865,Z 210.971,A -85,B 0,C 180,E1 -5572.073,E2 -5572.073} C_VEL
LIN {X 0,Y 509.928,Z 210.961,A -85,B 0,C 180,E1 -5574.46,E2 -5574.46} C_VEL
LIN {X 0,Y 510.024,Z 210.957,A -85,B 0,C 180,E1 -5577.626,E2 -5577.626} C_VEL
LIN {X 0,Y 510.013,Z 210.953,A -85,B 0,C 180,E1 -5579.996,E2 -5579.996} C_VEL
LIN {X 0,Y 510.026,Z 210.949,A -85,B 0,C 180,E1 -5582.365,E2 -5582.365} C_VEL
LIN {X 0,Y 509.914,Z 210.971,A -85,B 0,C 180,E1 -5585.532,E2 -5585.532} C_VEL
LIN {X 0,Y 509.86,Z 210.972,A -85,B 0,C 180,E1 -5587.918,E2 -5587.918} C_VEL
LIN {X 0,Y 509.885,Z 210.97,A -85,B 0,C 180,E1 -5591.121,E2 -5591.121} C_VEL
LIN {X 0,Y 509.818,Z 210.975,A -85,B 0,C 180,E1 -5594.362,E2 -5594.362} C_VEL
LIN {X 0,Y 509.831,Z 210.974,A -85,B 0,C 180,E1 -5596.821,E2 -5596.821} C_VEL
LIN {X 0,Y 509.886,Z 210.967,A -85,B 0,C 180,E1 -5600.151,E2 -5600.151} C_VEL
LIN {X 0,Y 509.786,Z 210.985,A -85,B 0,C 180,E1 -5603.559,E2 -5603.559} C_VEL
LIN {X 0,Y 509.845,Z 210.971,A -85,B 0,C 180,E1 -5606.366,E2 -5606.366} C_VEL
LIN {X 0,Y 509.835,Z 210.975,A -85,B 0,C 180,E1 -5608.84,E2 -5608.84} C_VEL
LIN {X 0,Y 509.78,Z 210.985,A -85,B 0,C 180,E1 -5611.586,E2 -5611.586} C_VEL
LIN {X 0,Y 509.806,Z 210.976,A -85,B 0,C 180,E1 -5614.409,E2 -5614.409} C_VEL
LIN {X 0,Y 509.772,Z 210.989,A -85,B 0,C 180,E1 -5617.336,E2 -5617.336} C_VEL
LIN {X 0,Y 509.792,Z 210.978,A -85,B 0,C 180,E1 -5620.378,E2 -5620.378} C_VEL
LIN {X 0,Y 509.777,Z 210.985,A -85,B 0,C 180,E1 -5623.058,E2 -5623.058} C_VEL
LIN {X 0,Y 509.781,Z 210.981,A -85,B 0,C 180,E1 -5625.788,E2 -5625.788} C_VEL
LIN {X 0,Y 509.812,Z 210.976,A -85,B 0,C 180,E1 -5628.571,E2 -5628.571} C_VEL
LIN {X 0,Y 509.799,Z 210.979,A -85,B 0,C 180,E1 -5631.782,E2 -5631.782} C_VEL
LIN {X 0,Y 509.784,Z 210.982,A -85,B 0,C 180,E1 -5633.686,E2 -5633.686} C_VEL
LIN {X 0,Y 509.115,Z 211.063,A -85,B 0,C 180,E1 -5634.345,E2 -5634.345} C_VEL
LIN {X 0,Y 506.298,Z 211.419,A -85,B 0,C 180,E1 -5635.417,E2 -5635.417} C_VEL
LIN {X 0,Y 503.906,Z 211.719,A -85,B 0,C 180,E1 -5636.281,E2 -5636.281} C_VEL
LIN {X 0,Y 502.855,Z 211.847,A -85,B 0,C 180,E1 -5636.947,E2 -5636.947} C_VEL
LIN {X 0,Y 502.756,Z 211.858,A -85,B 0,C 180,E1 -5637.172,E2 -5637.172} C_VEL
LIN {X 0,Y 502.772,Z 211.852,A -85,B 0,C 180,E1 -5640.059,E2 -5640.059} C_VEL
LIN {X 0,Y 502.775,Z 211.853,A -85,B 0,C 180,E1 -5642.531,E2 -5642.531} C_VEL
LIN {X 0,Y 502.775,Z 211.859,A -85,B 0,C 180,E1 -5645.294,E2 -5645.294} C_VEL
LIN {X 0,Y 502.759,Z 211.855,A -85,B 0,C 180,E1 -5647.826,E2 -5647.826} C_VEL
LIN {X 0,Y 502.763,Z 211.854,A -85,B 0,C 180,E1 -5650.398,E2 -5650.398} C_VEL
LIN {X 0,Y 502.784,Z 211.857,A -85,B 0,C 180,E1 -5652.93,E2 -5652.93} C_VEL
LIN {X 0,Y 502.78,Z 211.856,A -85,B 0,C 180,E1 -5655.428,E2 -5655.428} C_VEL
LIN {X 0,Y 502.836,Z 211.848,A -85,B 0,C 180,E1 -5658.716,E2 -5658.716} C_VEL
LIN {X 0,Y 502.852,Z 211.842,A -85,B 0,C 180,E1 -5661.966,E2 -5661.966} C_VEL
LIN {X 0,Y 502.9,Z 211.837,A -85,B 0,C 180,E1 -5664.386,E2 -5664.386} C_VEL
LIN {X 0,Y 502.962,Z 211.831,A -85,B 0,C 180,E1 -5667.597,E2 -5667.597} C_VEL
LIN {X 0,Y 502.957,Z 211.829,A -85,B 0,C 180,E1 -5670,E2 -5670} C_VEL
LIN {X 0,Y 502.962,Z 211.83,A -85,B 0,C 180,E1 -5672.402,E2 -5672.402} C_VEL
LIN {X 0,Y 502.9,Z 211.838,A -85,B 0,C 180,E1 -5675.614,E2 -5675.614} C_VEL
LIN {X 0,Y 502.852,Z 211.844,A -85,B 0,C 180,E1 -5678.034,E2 -5678.034} C_VEL
LIN {X 0,Y 502.835,Z 211.852,A -85,B 0,C 180,E1 -5681.284,E2 -5681.284} C_VEL
LIN {X 0,Y 502.857,Z 211.892,A -85,B 0,C 180,E1 -5682.87,E2 -5682.87} C_VEL
LIN {X 0,Y 503.556,Z 218.122,A -85,B 0,C 180,E1 -5684.137,E2 -5684.137} C_VEL
LIN {X 0,Y 503.284,Z 231.95,A -85,B 0,C 180,E1 -5686.843,E2 -5686.843} C_VEL
LIN {X 0,Y 503.258,Z 234.249,A -85,B 0,C 180,E1 -5687.262,E2 -5687.262} C_VEL
LIN {X 0,Y 505.424,Z 245.6,A -85,B 0,C 180,E1 -5687.499,E2 -5687.499} C_VEL
LIN {X 0,Y 504.827,Z 341.691,A -85,B 0,C 180,E1 -5688.907,E2 -5688.907} C_VEL
LIN {X 0,Y 504.588,Z 355.262,A -85,B 0,C 180,E1 -5689.281,E2 -5689.281} C_VEL
LIN {X 0,Y 504.35,Z 367.932,A -85,B 0,C 180,E1 -5689.802,E2 -5689.802} C_VEL
LIN {X 0,Y 504.053,Z 379.785,A -85,B 0,C 180,E1 -5690.466,E2 -5690.466} C_VEL
LIN {X 0,Y 503.69,Z 391.036,A -85,B 0,C 180,E1 -5691.27,E2 -5691.27} C_VEL
LIN {X 0,Y 503.308,Z 400.92,A -85,B 0,C 180,E1 -5692.148,E2 -5692.148} C_VEL
LIN {X 0,Y 502.946,Z 410.869,A -85,B 0,C 180,E1 -5693.25,E2 -5693.25} C_VEL
LIN {X 0,Y 502.693,Z 420.035,A -85,B 0,C 180,E1 -5694.516,E2 -5694.516} C_VEL
LIN {X 0,Y 502.459,Z 426.865,A -85,B 0,C 180,E1 -5695.696,E2 -5695.696} C_VEL
LIN {X 0,Y 502.292,Z 433.036,A -85,B 0,C 180,E1 -5697.047,E2 -5697.047} C_VEL
LIN {X 0,Y 502.214,Z 437.795,A -85,B 0,C 180,E1 -5698.41,E2 -5698.41} C_VEL
LIN {X 0,Y 502.067,Z 441.295,A -85,B 0,C 180,E1 -5699.802,E2 -5699.802} C_VEL
LIN {X 0,Y 501.996,Z 443.66,A -85,B 0,C 180,E1 -5701.364,E2 -5701.364} C_VEL
LIN {X 0,Y 501.989,Z 444.529,A -85,B 0,C 180,E1 -5702.872,E2 -5702.872} C_VEL
LIN {X 0,Y 502.01,Z 444.061,A -85,B 0,C 180,E1 -5704.325,E2 -5704.325} C_VEL
LIN {X 0,Y 502.018,Z 442.351,A -85,B 0,C 180,E1 -5705.724,E2 -5705.724} C_VEL
LIN {X 0,Y 502.164,Z 439.447,A -85,B 0,C 180,E1 -5707.097,E2 -5707.097} C_VEL
LIN {X 0,Y 502.217,Z 435.457,A -85,B 0,C 180,E1 -5708.415,E2 -5708.415} C_VEL
LIN {X 0,Y 502.422,Z 430.218,A -85,B 0,C 180,E1 -5709.715,E2 -5709.715} C_VEL
LIN {X 0,Y 502.596,Z 423.103,A -85,B 0,C 180,E1 -5711.087,E2 -5711.087} C_VEL
LIN {X 0,Y 502.799,Z 415.784,A -85,B 0,C 180,E1 -5712.209,E2 -5712.209} C_VEL
LIN {X 0,Y 503.153,Z 406.471,A -85,B 0,C 180,E1 -5713.367,E2 -5713.367} C_VEL
LIN {X 0,Y 503.512,Z 396.66,A -85,B 0,C 180,E1 -5714.353,E2 -5714.353} C_VEL
LIN {X 0,Y 503.847,Z 385.563,A -85,B 0,C 180,E1 -5715.244,E2 -5715.244} C_VEL
LIN {X 0,Y 504.215,Z 373.784,A -85,B 0,C 180,E1 -5715.99,E2 -5715.99} C_VEL
LIN {X 0,Y 504.513,Z 361.12,A -85,B 0,C 180,E1 -5716.595,E2 -5716.595} C_VEL
LIN {X 0,Y 504.776,Z 347.802,A -85,B 0,C 180,E1 -5717.039,E2 -5717.039} C_VEL
LIN {X 0,Y 504.949,Z 334.876,A -85,B 0,C 180,E1 -5717.305,E2 -5717.305} C_VEL
LIN {X 0,Y 505.394,Z 245.287,A -85,B 0,C 180,E1 -5718.602,E2 -5718.602} C_VEL
LIN {X 0,Y 503.259,Z 233.947,A -85,B 0,C 180,E1 -5718.854,E2 -5718.854} C_VEL
LIN {X 0,Y 503.477,Z 217.973,A -85,B 0,C 180,E1 -5721.771,E2 -5721.771} C_VEL
LIN {X 0,Y 502.933,Z 212.487,A -85,B 0,C 180,E1 -5722.797,E2 -5722.797} C_VEL
LIN {X 0,Y 502.814,Z 211.856,A -85,B 0,C 180,E1 -5722.973,E2 -5722.973} C_VEL
LIN {X 0,Y 502.772,Z 211.856,A -85,B 0,C 180,E1 -5726.011,E2 -5726.011} C_VEL
LIN {X 0,Y 502.762,Z 211.862,A -85,B 0,C 180,E1 -5728.862,E2 -5728.862} C_VEL
LIN {X 0,Y 502.811,Z 211.85,A -85,B 0,C 180,E1 -5731.709,E2 -5731.709} C_VEL
LIN {X 0,Y 502.809,Z 211.849,A -85,B 0,C 180,E1 -5734.329,E2 -5734.329} C_VEL
LIN {X 0,Y 502.774,Z 211.857,A -85,B 0,C 180,E1 -5737.302,E2 -5737.302} C_VEL
LIN {X 0,Y 502.798,Z 211.853,A -85,B 0,C 180,E1 -5740.405,E2 -5740.405} C_VEL
LIN {X 0,Y 502.808,Z 211.856,A -85,B 0,C 180,E1 -5742.937,E2 -5742.937} C_VEL
LIN {X 0,Y 502.82,Z 211.849,A -85,B 0,C 180,E1 -5745.434,E2 -5745.434} C_VEL
LIN {X 0,Y 502.877,Z 211.845,A -85,B 0,C 180,E1 -5748.722,E2 -5748.722} C_VEL
LIN {X 0,Y 502.862,Z 211.841,A -85,B 0,C 180,E1 -5751.971,E2 -5751.971} C_VEL
LIN {X 0,Y 502.91,Z 211.839,A -85,B 0,C 180,E1 -5754.391,E2 -5754.391} C_VEL
LIN {X 0,Y 503.004,Z 211.823,A -85,B 0,C 180,E1 -5757.602,E2 -5757.602} C_VEL
LIN {X 0,Y 503.021,Z 211.828,A -85,B 0,C 180,E1 -5760.805,E2 -5760.805} C_VEL
LIN {X 0,Y 502.848,Z 211.846,A -85,B 0,C 180,E1 -5763.209,E2 -5763.209} C_VEL
LIN {X 0,Y 502.88,Z 211.842,A -85,B 0,C 180,E1 -5766.423,E2 -5766.423} C_VEL
LIN {X 0,Y 502.84,Z 211.849,A -85,B 0,C 180,E1 -5768.848,E2 -5768.848} C_VEL
LIN {X 0,Y 502.839,Z 211.846,A -85,B 0,C 180,E1 -5772.106,E2 -5772.106} C_VEL
LIN {X 0,Y 502.845,Z 211.844,A -85,B 0,C 180,E1 -5775.404,E2 -5775.404} C_VEL
LIN {X 0,Y 502.819,Z 211.852,A -85,B 0,C 180,E1 -5778.756,E2 -5778.756} C_VEL
LIN {X 0,Y 502.781,Z 211.851,A -85,B 0,C 180,E1 -5781.315,E2 -5781.315} C_VEL
LIN {X 0,Y 502.755,Z 211.855,A -85,B 0,C 180,E1 -5783.919,E2 -5783.919} C_VEL
LIN {X 0,Y 502.757,Z 211.86,A -85,B 0,C 180,E1 -5786.576,E2 -5786.576} C_VEL
LIN {X 0,Y 502.811,Z 211.847,A -85,B 0,C 180,E1 -5789.292,E2 -5789.292} C_VEL
LIN {X 0,Y 502.779,Z 211.856,A -85,B 0,C 180,E1 -5792.088,E2 -5792.088} C_VEL
LIN {X 0,Y 502.783,Z 211.854,A -85,B 0,C 180,E1 -5794.97,E2 -5794.97} C_VEL
LIN {X 0,Y 502.758,Z 211.862,A -85,B 0,C 180,E1 -5798.483,E2 -5798.483} C_VEL
LIN {X 0,Y 502.758,Z 211.857,A -85,B 0,C 180,E1 -5801.075,E2 -5801.075} C_VEL
LIN {X 0,Y 502.782,Z 211.859,A -85,B 0,C 180,E1 -5804.531,E2 -5804.531} C_VEL
LIN {X 0,Y 502.736,Z 211.861,A -85,B 0,C 180,E1 -5807.856,E2 -5807.856} C_VEL
LIN {X 0,Y 502.767,Z 211.855,A -85,B 0,C 180,E1 -5811.022,E2 -5811.022} C_VEL
LIN {X 0,Y 502.746,Z 211.864,A -85,B 0,C 180,E1 -5814.177,E2 -5814.177} C_VEL
LIN {X 0,Y 502.775,Z 211.856,A -85,B 0,C 180,E1 -5817.007,E2 -5817.007} C_VEL
LIN {X 0,Y 502.751,Z 211.867,A -85,B 0,C 180,E1 -5820.081,E2 -5820.081} C_VEL
LIN {X 0,Y 502.743,Z 211.863,A -85,B 0,C 180,E1 -5822.529,E2 -5822.529} C_VEL
LIN {X 0,Y 502.797,Z 212.042,A -85,B 0,C 180,E1 -5825.098,E2 -5825.098} C_VEL
LIN {X 0,Y 504.379,Z 220.613,A -85,B 0,C 180,E1 -5826.572,E2 -5826.572} C_VEL
LIN {X 0,Y 504.041,Z 236.334,A -85,B 0,C 180,E1 -5829.103,E2 -5829.103} C_VEL
LIN {X 0,Y 503.568,Z 255.337,A -85,B 0,C 180,E1 -5832.12,E2 -5832.12} C_VEL
LIN {X 0,Y 503.238,Z 268.751,A -85,B 0,C 180,E1 -5834.196,E2 -5834.196} C_VEL
LIN {X 0,Y 505.309,Z 282.874,A -85,B 0,C 180,E1 -5834.469,E2 -5834.469} C_VEL
LIN {X 0,Y 504.818,Z 377.192,A -85,B 0,C 180,E1 -5835.848,E2 -5835.848} C_VEL
LIN {X 0,Y 504.509,Z 390.392,A -85,B 0,C 180,E1 -5836.199,E2 -5836.199} C_VEL
LIN {X 0,Y 504.183,Z 403.104,A -85,B 0,C 180,E1 -5836.703,E2 -5836.703} C_VEL
LIN {X 0,Y 503.871,Z 414.15,A -85,B 0,C 180,E1 -5837.294,E2 -5837.294} C_VEL
LIN {X 0,Y 503.513,Z 426.106,A -85,B 0,C 180,E1 -5838.119,E2 -5838.119} C_VEL
LIN {X 0,Y 503.206,Z 436.631,A -85,B 0,C 180,E1 -5839.03,E2 -5839.03} C_VEL
LIN {X 0,Y 502.835,Z 445.232,A -85,B 0,C 180,E1 -5839.939,E2 -5839.939} C_VEL
LIN {X 0,Y 502.612,Z 453.172,A -85,B 0,C 180,E1 -5840.95,E2 -5840.95} C_VEL
LIN {X 0,Y 502.386,Z 460.926,A -85,B 0,C 180,E1 -5842.161,E2 -5842.161} C_VEL
LIN {X 0,Y 502.243,Z 468.071,A -85,B 0,C 180,E1 -5843.573,E2 -5843.573} C_VEL
LIN {X 0,Y 502.173,Z 472.827,A -85,B 0,C 180,E1 -5844.781,E2 -5844.781} C_VEL
LIN {X 0,Y 502.14,Z 476.461,A -85,B 0,C 180,E1 -5845.987,E2 -5845.987} C_VEL
LIN {X 0,Y 502.123,Z 478.337,A -85,B 0,C 180,E1 -5846.791,E2 -5846.791} C_VEL
LIN {X 0,Y 502.094,Z 479.743,A -85,B 0,C 180,E1 -5847.593,E2 -5847.593} C_VEL
LIN {X 0,Y 501.994,Z 481.361,A -85,B 0,C 180,E1 -5849.198,E2 -5849.198} C_VEL
LIN {X 0,Y 501.987,Z 481.582,A -85,B 0,C 180,E1 -5850,E2 -5850} C_VEL
LIN {X 0,Y 502.038,Z 480.763,A -85,B 0,C 180,E1 -5851.604,E2 -5851.604} C_VEL
LIN {X 0,Y 502.094,Z 479.769,A -85,B 0,C 180,E1 -5852.407,E2 -5852.407} C_VEL
LIN {X 0,Y 502.123,Z 478.369,A -85,B 0,C 180,E1 -5853.209,E2 -5853.209} C_VEL
LIN {X 0,Y 502.103,Z 475.423,A -85,B 0,C 180,E1 -5854.415,E2 -5854.415} C_VEL
LIN {X 0,Y 502.201,Z 471.437,A -85,B 0,C 180,E1 -5855.622,E2 -5855.622} C_VEL
LIN {X 0,Y 502.278,Z 465.399,A -85,B 0,C 180,E1 -5857.012,E2 -5857.012} C_VEL
LIN {X 0,Y 502.482,Z 458.593,A -85,B 0,C 180,E1 -5858.242,E2 -5858.242} C_VEL
LIN {X 0,Y 502.715,Z 450.274,A -85,B 0,C 180,E1 -5859.454,E2 -5859.454} C_VEL
LIN {X 0,Y 502.969,Z 441.735,A -85,B 0,C 180,E1 -5860.466,E2 -5860.466} C_VEL
LIN {X 0,Y 503.39,Z 431.192,A -85,B 0,C 180,E1 -5861.475,E2 -5861.475} C_VEL
LIN {X 0,Y 503.69,Z 419.366,A -85,B 0,C 180,E1 -5862.384,E2 -5862.384} C_VEL
LIN {X 0,Y 504.082,Z 407.336,A -85,B 0,C 180,E1 -5863.094,E2 -5863.094} C_VEL
LIN {X 0,Y 504.39,Z 394.87,A -85,B 0,C 180,E1 -5863.65,E2 -5863.65} C_VEL
LIN {X 0,Y 504.682,Z 381.956,A -85,B 0,C 180,E1 -5864.053,E2 -5864.053} C_VEL
LIN {X 0,Y 504.916,Z 366.432,A -85,B 0,C 180,E1 -5864.329,E2 -5864.329} C_VEL
LIN {X 0,Y 505.202,Z 281.724,A -85,B 0,C 180,E1 -5865.554,E2 -5865.554} C_VEL
LIN {X 0,Y 503.256,Z 268.728,A -85,B 0,C 180,E1 -5865.822,E2 -5865.822} C_VEL
LIN {X 0,Y 503.776,Z 249.281,A -85,B 0,C 180,E1 -5868.926,E2 -5868.926} C_VEL
LIN {X 0,Y 504.31,Z 231,A -85,B 0,C 180,E1 -5871.887,E2 -5871.887} C_VEL
LIN {X 0,Y 504.554,Z 221.525,A -85,B 0,C 180,E1 -5873.441,E2 -5873.441} C_VEL
LIN {X 0,Y 502.775,Z 211.86,A -85,B 0,C 180,E1 -5875.174,E2 -5875.174} C_VEL
LIN {X 0,Y 502.756,Z 211.859,A -85,B 0,C 180,E1 -5878.377,E2 -5878.377} C_VEL
LIN {X 0,Y 502.766,Z 211.859,A -85,B 0,C 180,E1 -5881.491,E2 -5881.491} C_VEL
LIN {X 0,Y 502.771,Z 211.854,A -85,B 0,C 180,E1 -5884.436,E2 -5884.436} C_VEL
LIN {X 0,Y 502.744,Z 211.862,A -85,B 0,C 180,E1 -5887.957,E2 -5887.957} C_VEL
LIN {X 0,Y 502.753,Z 211.856,A -85,B 0,C 180,E1 -5891.071,E2 -5891.071} C_VEL
LIN {X 0,Y 502.754,Z 211.855,A -85,B 0,C 180,E1 -5894.523,E2 -5894.523} C_VEL
LIN {X 0,Y 502.75,Z 211.863,A -85,B 0,C 180,E1 -5897.806,E2 -5897.806} C_VEL
LIN {X 0,Y 502.762,Z 211.854,A -85,B 0,C 180,E1 -5901.017,E2 -5901.017} C_VEL
LIN {X 0,Y 502.712,Z 211.862,A -85,B 0,C 180,E1 -5904.177,E2 -5904.177} C_VEL
LIN {X 0,Y 502.769,Z 211.854,A -85,B 0,C 180,E1 -5907.002,E2 -5907.002} C_VEL
LIN {X 0,Y 502.745,Z 211.859,A -85,B 0,C 180,E1 -5910.076,E2 -5910.076} C_VEL
LIN {X 0,Y 502.738,Z 211.857,A -85,B 0,C 180,E1 -5912.524,E2 -5912.524} C_VEL
LIN {X 0,Y 502.763,Z 211.858,A -85,B 0,C 180,E1 -5915.312,E2 -5915.312} C_VEL
LIN {X 0,Y 502.771,Z 211.858,A -85,B 0,C 180,E1 -5917.823,E2 -5917.823} C_VEL
LIN {X 0,Y 502.769,Z 211.853,A -85,B 0,C 180,E1 -5920.394,E2 -5920.394} C_VEL
LIN {X 0,Y 502.769,Z 211.854,A -85,B 0,C 180,E1 -5922.926,E2 -5922.926} C_VEL
LIN {X 0,Y 502.82,Z 211.853,A -85,B 0,C 180,E1 -5925.425,E2 -5925.425} C_VEL
LIN {X 0,Y 502.825,Z 211.846,A -85,B 0,C 180,E1 -5928.712,E2 -5928.712} C_VEL
LIN {X 0,Y 502.837,Z 211.847,A -85,B 0,C 180,E1 -5931.962,E2 -5931.962} C_VEL
LIN {X 0,Y 502.884,Z 211.839,A -85,B 0,C 180,E1 -5934.382,E2 -5934.382} C_VEL
LIN {X 0,Y 502.992,Z 211.833,A -85,B 0,C 180,E1 -5937.593,E2 -5937.593} C_VEL
LIN {X 0,Y 502.983,Z 211.828,A -85,B 0,C 180,E1 -5939.995,E2 -5939.995} C_VEL
LIN {X 0,Y 502.995,Z 211.825,A -85,B 0,C 180,E1 -5942.398,E2 -5942.398} C_VEL
LIN {X 0,Y 502.869,Z 211.847,A -85,B 0,C 180,E1 -5945.609,E2 -5945.609} C_VEL
LIN {X 0,Y 502.831,Z 211.847,A -85,B 0,C 180,E1 -5948.029,E2 -5948.029} C_VEL
LIN {X 0,Y 502.851,Z 211.849,A -85,B 0,C 180,E1 -5951.278,E2 -5951.278} C_VEL
LIN {X 0,Y 502.799,Z 211.849,A -85,B 0,C 180,E1 -5954.567,E2 -5954.567} C_VEL
LIN {X 0,Y 502.79,Z 211.853,A -85,B 0,C 180,E1 -5957.904,E2 -5957.904} C_VEL
LIN {X 0,Y 502.801,Z 211.849,A -85,B 0,C 180,E1 -5960.531,E2 -5960.531} C_VEL
LIN {X 0,Y 502.755,Z 211.858,A -85,B 0,C 180,E1 -5963.036,E2 -5963.036} C_VEL
LIN {X 0,Y 502.802,Z 211.849,A -85,B 0,C 180,E1 -5966.563,E2 -5966.563} C_VEL
LIN {X 0,Y 502.785,Z 211.859,A -85,B 0,C 180,E1 -5969.283,E2 -5969.283} C_VEL
LIN {X 0,Y 502.744,Z 211.856,A -85,B 0,C 180,E1 -5972.08,E2 -5972.08} C_VEL
LIN {X 0,Y 502.757,Z 211.858,A -85,B 0,C 180,E1 -5974.961,E2 -5974.961} C_VEL
LIN {X 0,Y 502.749,Z 211.856,A -85,B 0,C 180,E1 -5977.95,E2 -5977.95} C_VEL
LIN {X 0,Y 502.774,Z 211.858,A -85,B 0,C 180,E1 -5981.061,E2 -5981.061} C_VEL
LIN {X 0,Y 502.752,Z 211.855,A -85,B 0,C 180,E1 -5984.527,E2 -5984.527} C_VEL
LIN {X 0,Y 502.747,Z 211.857,A -85,B 0,C 180,E1 -5987.857,E2 -5987.857} C_VEL
LIN {X 0,Y 502.737,Z 211.857,A -85,B 0,C 180,E1 -5990.241,E2 -5990.241} C_VEL
LIN {X 0,Y 502.729,Z 211.864,A -85,B 0,C 180,E1 -5993.05,E2 -5993.05} C_VEL
LIN {X 0,Y 502.752,Z 211.855,A -85,B 0,C 180,E1 -5996.003,E2 -5996.003} C_VEL
LIN {X 0,Y 502.756,Z 211.858,A -85,B 0,C 180,E1 -5997.172,E2 -5997.172} C_VEL
LIN {X 0,Y 502.054,Z 211.944,A -85,B 0,C 180,E1 -5997.841,E2 -5997.841} C_VEL
LIN {X 0,Y 499.196,Z 212.303,A -85,B 0,C 180,E1 -5998.927,E2 -5998.927} C_VEL
LIN {X 0,Y 496.806,Z 212.597,A -85,B 0,C 180,E1 -5999.802,E2 -5999.802} C_VEL
LIN {X 0,Y 495.786,Z 212.723,A -85,B 0,C 180,E1 -6000.478,E2 -6000.478} C_VEL
LIN {X 0,Y 495.706,Z 212.735,A -85,B 0,C 180,E1 -6000.707,E2 -6000.707} C_VEL
LIN {X 0,Y 495.739,Z 212.729,A -85,B 0,C 180,E1 -6003.93,E2 -6003.93} C_VEL
LIN {X 0,Y 495.727,Z 212.739,A -85,B 0,C 180,E1 -6007.129,E2 -6007.129} C_VEL
LIN {X 0,Y 495.715,Z 212.731,A -85,B 0,C 180,E1 -6010.108,E2 -6010.108} C_VEL
LIN {X 0,Y 495.737,Z 212.731,A -85,B 0,C 180,E1 -6012.68,E2 -6012.68} C_VEL
LIN {X 0,Y 495.725,Z 212.738,A -85,B 0,C 180,E1 -6015.216,E2 -6015.216} C_VEL
LIN {X 0,Y 495.809,Z 212.722,A -85,B 0,C 180,E1 -6018.554,E2 -6018.554} C_VEL
LIN {X 0,Y 495.82,Z 212.719,A -85,B 0,C 180,E1 -6021.851,E2 -6021.851} C_VEL
LIN {X 0,Y 495.856,Z 212.714,A -85,B 0,C 180,E1 -6024.306,E2 -6024.306} C_VEL
LIN {X 0,Y 495.932,Z 212.707,A -85,B 0,C 180,E1 -6027.563,E2 -6027.563} C_VEL
LIN {X 0,Y 495.928,Z 212.705,A -85,B 0,C 180,E1 -6030,E2 -6030} C_VEL
LIN {X 0,Y 495.932,Z 212.706,A -85,B 0,C 180,E1 -6032.436,E2 -6032.436} C_VEL
LIN {X 0,Y 495.856,Z 212.715,A -85,B 0,C 180,E1 -6035.694,E2 -6035.694} C_VEL
LIN {X 0,Y 495.821,Z 212.72,A -85,B 0,C 180,E1 -6038.149,E2 -6038.149} C_VEL
LIN {X 0,Y 495.812,Z 212.726,A -85,B 0,C 180,E1 -6041.446,E2 -6041.446} C_VEL
LIN {X 0,Y 495.833,Z 212.84,A -85,B 0,C 180,E1 -6042.743,E2 -6042.743} C_VEL
LIN {X 0,Y 496.597,Z 219.594,A -85,B 0,C 180,E1 -6044.13,E2 -6044.13} C_VEL
LIN {X 0,Y 496.298,Z 233.505,A -85,B 0,C 180,E1 -6046.875,E2 -6046.875} C_VEL
LIN {X 0,Y 496.283,Z 234.444,A -85,B 0,C 180,E1 -6047.035,E2 -6047.035} C_VEL
LIN {X 0,Y 498.6,Z 246.79,A -85,B 0,C 180,E1 -6047.297,E2 -6047.297} C_VEL
LIN {X 0,Y 497.972,Z 341.441,A -85,B 0,C 180,E1 -6048.701,E2 -6048.701} C_VEL
LIN {X 0,Y 497.73,Z 354.527,A -85,B 0,C 180,E1 -6049.058,E2 -6049.058} C_VEL
LIN {X 0,Y 497.469,Z 366.732,A -85,B 0,C 180,E1 -6049.55,E2 -6049.55} C_VEL
LIN {X 0,Y 497.196,Z 377.888,A -85,B 0,C 180,E1 -6050.154,E2 -6050.154} C_VEL
LIN {X 0,Y 496.822,Z 388.746,A -85,B 0,C 180,E1 -6050.905,E2 -6050.905} C_VEL
LIN {X 0,Y 496.395,Z 399.301,A -85,B 0,C 180,E1 -6051.817,E2 -6051.817} C_VEL
LIN {X 0,Y 496.059,Z 409.129,A -85,B 0,C 180,E1 -6052.868,E2 -6052.868} C_VEL
LIN {X 0,Y 495.705,Z 418.038,A -85,B 0,C 180,E1 -6054.054,E2 -6054.054} C_VEL
LIN {X 0,Y 495.483,Z 426.139,A -85,B 0,C 180,E1 -6055.408,E2 -6055.408} C_VEL
LIN {X 0,Y 495.264,Z 431.986,A -85,B 0,C 180,E1 -6056.637,E2 -6056.637} C_VEL
LIN {X 0,Y 495.138,Z 436.791,A -85,B 0,C 180,E1 -6057.93,E2 -6057.93} C_VEL
LIN {X 0,Y 495.03,Z 440.615,A -85,B 0,C 180,E1 -6059.327,E2 -6059.327} C_VEL
LIN {X 0,Y 494.926,Z 443.199,A -85,B 0,C 180,E1 -6060.743,E2 -6060.743} C_VEL
LIN {X 0,Y 494.906,Z 444.268,A -85,B 0,C 180,E1 -6061.696,E2 -6061.696} C_VEL
LIN {X 0,Y 494.891,Z 444.815,A -85,B 0,C 180,E1 -6063.098,E2 -6063.098} C_VEL
LIN {X 0,Y 494.911,Z 444.072,A -85,B 0,C 180,E1 -6064.611,E2 -6064.611} C_VEL
LIN {X 0,Y 494.94,Z 442.234,A -85,B 0,C 180,E1 -6065.977,E2 -6065.977} C_VEL
LIN {X 0,Y 495.128,Z 438.5,A -85,B 0,C 180,E1 -6067.614,E2 -6067.614} C_VEL
LIN {X 0,Y 495.235,Z 433.235,A -85,B 0,C 180,E1 -6069.16,E2 -6069.16} C_VEL
LIN {X 0,Y 495.437,Z 427.028,A -85,B 0,C 180,E1 -6070.532,E2 -6070.532} C_VEL
LIN {X 0,Y 495.658,Z 419.762,A -85,B 0,C 180,E1 -6071.79,E2 -6071.79} C_VEL
LIN {X 0,Y 496.054,Z 411.155,A -85,B 0,C 180,E1 -6072.985,E2 -6072.985} C_VEL
LIN {X 0,Y 496.368,Z 401.535,A -85,B 0,C 180,E1 -6074.07,E2 -6074.07} C_VEL
LIN {X 0,Y 496.748,Z 390.952,A -85,B 0,C 180,E1 -6075.022,E2 -6075.022} C_VEL
LIN {X 0,Y 497.141,Z 379.534,A -85,B 0,C 180,E1 -6075.842,E2 -6075.842} C_VEL
LIN {X 0,Y 497.483,Z 368.016,A -85,B 0,C 180,E1 -6076.488,E2 -6076.488} C_VEL
LIN {X 0,Y 497.784,Z 355.27,A -85,B 0,C 180,E1 -6077.013,E2 -6077.013} C_VEL
LIN {X 0,Y 497.972,Z 341.946,A -85,B 0,C 180,E1 -6077.383,E2 -6077.383} C_VEL
LIN {X 0,Y 498.596,Z 246.205,A -85,B 0,C 180,E1 -6078.811,E2 -6078.811} C_VEL
LIN {X 0,Y 496.292,Z 234.15,A -85,B 0,C 180,E1 -6079.083,E2 -6079.083} C_VEL
LIN {X 0,Y 496.496,Z 218.346,A -85,B 0,C 180,E1 -6082.002,E2 -6082.002} C_VEL
LIN {X 0,Y 495.789,Z 212.731,A -85,B 0,C 180,E1 -6083.074,E2 -6083.074} C_VEL
LIN {X 0,Y 495.724,Z 212.735,A -85,B 0,C 180,E1 -6086.441,E2 -6086.441} C_VEL
LIN {X 0,Y 495.72,Z 212.739,A -85,B 0,C 180,E1 -6089.318,E2 -6089.318} C_VEL
LIN {X 0,Y 495.748,Z 212.729,A -85,B 0,C 180,E1 -6092.114,E2 -6092.114} C_VEL
LIN {X 0,Y 495.757,Z 212.733,A -85,B 0,C 180,E1 -6094.838,E2 -6094.838} C_VEL
LIN {X 0,Y 495.719,Z 212.734,A -85,B 0,C 180,E1 -6097.5,E2 -6097.5} C_VEL
LIN {X 0,Y 495.744,Z 212.73,A -85,B 0,C 180,E1 -6100.115,E2 -6100.115} C_VEL
LIN {X 0,Y 495.76,Z 212.733,A -85,B 0,C 180,E1 -6102.686,E2 -6102.686} C_VEL
LIN {X 0,Y 495.765,Z 212.73,A -85,B 0,C 180,E1 -6105.222,E2 -6105.222} C_VEL
LIN {X 0,Y 495.851,Z 212.719,A -85,B 0,C 180,E1 -6108.56,E2 -6108.56} C_VEL
LIN {X 0,Y 495.818,Z 212.718,A -85,B 0,C 180,E1 -6111.856,E2 -6111.856} C_VEL
LIN {X 0,Y 495.867,Z 212.715,A -85,B 0,C 180,E1 -6114.311,E2 -6114.311} C_VEL
LIN {X 0,Y 495.974,Z 212.699,A -85,B 0,C 180,E1 -6117.568,E2 -6117.568} C_VEL
LIN {X 0,Y 495.971,Z 212.706,A -85,B 0,C 180,E1 -6120.816,E2 -6120.816} C_VEL
LIN {X 0,Y 495.969,Z 212.703,A -85,B 0,C 180,E1 -6122.441,E2 -6122.441} C_VEL
LIN {X 0,Y 495.867,Z 212.71,A -85,B 0,C 180,E1 -6125.698,E2 -6125.698} C_VEL
LIN {X 0,Y 495.82,Z 212.721,A -85,B 0,C 180,E1 -6128.153,E2 -6128.153} C_VEL
LIN {X 0,Y 495.842,Z 212.717,A -85,B 0,C 180,E1 -6131.449,E2 -6131.449} C_VEL
LIN {X 0,Y 495.782,Z 212.729,A -85,B 0,C 180,E1 -6134.787,E2 -6134.787} C_VEL
LIN {X 0,Y 495.754,Z 212.727,A -85,B 0,C 180,E1 -6137.324,E2 -6137.324} C_VEL
LIN {X 0,Y 495.765,Z 212.726,A -85,B 0,C 180,E1 -6139.894,E2 -6139.894} C_VEL
LIN {X 0,Y 495.756,Z 212.73,A -85,B 0,C 180,E1 -6142.863,E2 -6142.863} C_VEL
LIN {X 0,Y 495.706,Z 212.735,A -85,B 0,C 180,E1 -6146.076,E2 -6146.076} C_VEL
LIN {X 0,Y 495.742,Z 212.732,A -85,B 0,C 180,E1 -6148.82,E2 -6148.82} C_VEL
LIN {X 0,Y 495.75,Z 212.728,A -85,B 0,C 180,E1 -6151.727,E2 -6151.727} C_VEL
LIN {X 0,Y 495.756,Z 212.733,A -85,B 0,C 180,E1 -6154.694,E2 -6154.694} C_VEL
LIN {X 0,Y 495.7,Z 212.734,A -85,B 0,C 180,E1 -6157.567,E2 -6157.567} C_VEL
LIN {X 0,Y 495.714,Z 212.736,A -85,B 0,C 180,E1 -6160.043,E2 -6160.043} C_VEL
LIN {X 0,Y 495.694,Z 212.739,A -85,B 0,C 180,E1 -6162.89,E2 -6162.89} C_VEL
LIN {X 0,Y 495.717,Z 212.738,A -85,B 0,C 180,E1 -6165.999,E2 -6165.999} C_VEL
LIN {X 0,Y 495.712,Z 212.733,A -85,B 0,C 180,E1 -6169.296,E2 -6169.296} C_VEL
LIN {X 0,Y 495.711,Z 212.734,A -85,B 0,C 180,E1 -6171.406,E2 -6171.406} C_VEL
LIN {X 0,Y 495.719,Z 212.739,A -85,B 0,C 180,E1 -6174.461,E2 -6174.461} C_VEL
LIN {X 0,Y 495.73,Z 212.734,A -85,B 0,C 180,E1 -6177.404,E2 -6177.404} C_VEL
LIN {X 0,Y 495.702,Z 212.744,A -85,B 0,C 180,E1 -6180.25,E2 -6180.25} C_VEL
LIN {X 0,Y 495.701,Z 212.737,A -85,B 0,C 180,E1 -6183.283,E2 -6183.283} C_VEL
LIN {X 0,Y 495.745,Z 212.819,A -85,B 0,C 180,E1 -6184.902,E2 -6184.902} C_VEL
LIN {X 0,Y 497.446,Z 221.97,A -85,B 0,C 180,E1 -6186.5,E2 -6186.5} C_VEL
LIN {X 0,Y 497.072,Z 237.61,A -85,B 0,C 180,E1 -6189.053,E2 -6189.053} C_VEL
LIN {X 0,Y 496.51,Z 257.687,A -85,B 0,C 180,E1 -6192.283,E2 -6192.283} C_VEL
LIN {X 0,Y 496.23,Z 268.182,A -85,B 0,C 180,E1 -6193.955,E2 -6193.955} C_VEL
LIN {X 0,Y 498.47,Z 283.883,A -85,B 0,C 180,E1 -6194.268,E2 -6194.268} C_VEL
LIN {X 0,Y 497.944,Z 376.82,A -85,B 0,C 180,E1 -6195.648,E2 -6195.648} C_VEL
LIN {X 0,Y 497.605,Z 390.047,A -85,B 0,C 180,E1 -6196.004,E2 -6196.004} C_VEL
LIN {X 0,Y 497.26,Z 402.777,A -85,B 0,C 180,E1 -6196.515,E2 -6196.515} C_VEL
LIN {X 0,Y 496.915,Z 414.15,A -85,B 0,C 180,E1 -6197.133,E2 -6197.133} C_VEL
LIN {X 0,Y 496.506,Z 425.8,A -85,B 0,C 180,E1 -6197.949,E2 -6197.949} C_VEL
LIN {X 0,Y 496.19,Z 436.332,A -85,B 0,C 180,E1 -6198.873,E2 -6198.873} C_VEL
LIN {X 0,Y 495.816,Z 444.939,A -85,B 0,C 180,E1 -6199.795,E2 -6199.795} C_VEL
LIN {X 0,Y 495.545,Z 452.883,A -85,B 0,C 180,E1 -6200.819,E2 -6200.819} C_VEL
LIN {X 0,Y 495.33,Z 460.645,A -85,B 0,C 180,E1 -6202.049,E2 -6202.049} C_VEL
LIN {X 0,Y 495.175,Z 465.959,A -85,B 0,C 180,E1 -6203.071,E2 -6203.071} C_VEL
LIN {X 0,Y 495.117,Z 471.113,A -85,B 0,C 180,E1 -6204.298,E2 -6204.298} C_VEL
LIN {X 0,Y 495.009,Z 475.112,A -85,B 0,C 180,E1 -6205.522,E2 -6205.522} C_VEL
LIN {X 0,Y 495.044,Z 478.071,A -85,B 0,C 180,E1 -6206.745,E2 -6206.745} C_VEL
LIN {X 0,Y 495.001,Z 479.479,A -85,B 0,C 180,E1 -6207.559,E2 -6207.559} C_VEL
LIN {X 0,Y 494.965,Z 480.484,A -85,B 0,C 180,E1 -6208.373,E2 -6208.373} C_VEL
LIN {X 0,Y 494.905,Z 481.321,A -85,B 0,C 180,E1 -6210,E2 -6210} C_VEL
LIN {X 0,Y 494.965,Z 480.503,A -85,B 0,C 180,E1 -6211.627,E2 -6211.627} C_VEL
LIN {X 0,Y 495.001,Z 479.508,A -85,B 0,C 180,E1 -6212.441,E2 -6212.441} C_VEL
LIN {X 0,Y 495.044,Z 478.108,A -85,B 0,C 180,E1 -6213.255,E2 -6213.255} C_VEL
LIN {X 0,Y 495.009,Z 475.16,A -85,B 0,C 180,E1 -6214.479,E2 -6214.479} C_VEL
LIN {X 0,Y 495.117,Z 471.172,A -85,B 0,C 180,E1 -6215.702,E2 -6215.702} C_VEL
LIN {X 0,Y 495.209,Z 465.03,A -85,B 0,C 180,E1 -6217.133,E2 -6217.133} C_VEL
LIN {X 0,Y 495.428,Z 458.322,A -85,B 0,C 180,E1 -6218.36,E2 -6218.36} C_VEL
LIN {X 0,Y 495.689,Z 450,A -85,B 0,C 180,E1 -6219.59,E2 -6219.59} C_VEL
LIN {X 0,Y 495.975,Z 441.454,A -85,B 0,C 180,E1 -6220.615,E2 -6220.615} C_VEL
LIN {X 0,Y 496.41,Z 430.901,A -85,B 0,C 180,E1 -6221.639,E2 -6221.639} C_VEL
LIN {X 0,Y 496.718,Z 419.205,A -85,B 0,C 180,E1 -6222.551,E2 -6222.551} C_VEL
LIN {X 0,Y 497.133,Z 407.014,A -85,B 0,C 180,E1 -6223.281,E2 -6223.281} C_VEL
LIN {X 0,Y 497.491,Z 394.526,A -85,B 0,C 180,E1 -6223.843,E2 -6223.843} C_VEL
LIN {X 0,Y 497.8,Z 381.553,A -85,B 0,C 180,E1 -6224.252,E2 -6224.252} C_VEL
LIN {X 0,Y 498.033,Z 365.939,A -85,B 0,C 180,E1 -6224.532,E2 -6224.532} C_VEL
LIN {X 0,Y 498.455,Z 283.343,A -85,B 0,C 180,E1 -6225.741,E2 -6225.741} C_VEL
LIN {X 0,Y 496.251,Z 268.563,A -85,B 0,C 180,E1 -6226.036,E2 -6226.036} C_VEL
LIN {X 0,Y 496.832,Z 249.039,A -85,B 0,C 180,E1 -6229.201,E2 -6229.201} C_VEL
LIN {X 0,Y 497.425,Z 230.75,A -85,B 0,C 180,E1 -6232.206,E2 -6232.206} C_VEL
LIN {X 0,Y 497.631,Z 223.036,A -85,B 0,C 180,E1 -6233.491,E2 -6233.491} C_VEL
LIN {X 0,Y 495.728,Z 212.737,A -85,B 0,C 180,E1 -6235.338,E2 -6235.338} C_VEL
LIN {X 0,Y 495.724,Z 212.735,A -85,B 0,C 180,E1 -6238.476,E2 -6238.476} C_VEL
LIN {X 0,Y 495.73,Z 212.737,A -85,B 0,C 180,E1 -6241.717,E2 -6241.717} C_VEL
LIN {X 0,Y 495.737,Z 212.729,A -85,B 0,C 180,E1 -6244.685,E2 -6244.685} C_VEL
LIN {X 0,Y 495.691,Z 212.74,A -85,B 0,C 180,E1 -6247.564,E2 -6247.564} C_VEL
LIN {X 0,Y 495.71,Z 212.737,A -85,B 0,C 180,E1 -6250.037,E2 -6250.037} C_VEL
LIN {X 0,Y 495.673,Z 212.737,A -85,B 0,C 180,E1 -6252.887,E2 -6252.887} C_VEL
LIN {X 0,Y 495.71,Z 212.737,A -85,B 0,C 180,E1 -6255.993,E2 -6255.993} C_VEL
LIN {X 0,Y 495.711,Z 212.735,A -85,B 0,C 180,E1 -6259.291,E2 -6259.291} C_VEL
LIN {X 0,Y 495.705,Z 212.737,A -85,B 0,C 180,E1 -6261.401,E2 -6261.401} C_VEL
LIN {X 0,Y 495.695,Z 212.734,A -85,B 0,C 180,E1 -6264.455,E2 -6264.455} C_VEL
LIN {X 0,Y 495.725,Z 212.735,A -85,B 0,C 180,E1 -6267.399,E2 -6267.399} C_VEL
LIN {X 0,Y 495.696,Z 212.735,A -85,B 0,C 180,E1 -6270.246,E2 -6270.246} C_VEL
LIN {X 0,Y 495.697,Z 212.737,A -85,B 0,C 180,E1 -6273.277,E2 -6273.277} C_VEL
LIN {X 0,Y 495.704,Z 212.741,A -85,B 0,C 180,E1 -6275.719,E2 -6275.719} C_VEL
LIN {X 0,Y 495.727,Z 212.731,A -85,B 0,C 180,E1 -6278.367,E2 -6278.367} C_VEL
LIN {X 0,Y 495.746,Z 212.729,A -85,B 0,C 180,E1 -6280.966,E2 -6280.966} C_VEL
LIN {X 0,Y 495.818,Z 212.719,A -85,B 0,C 180,E1 -6284.546,E2 -6284.546} C_VEL
LIN {X 0,Y 495.8,Z 212.724,A -85,B 0,C 180,E1 -6287.974,E2 -6287.974} C_VEL
LIN {X 0,Y 495.767,Z 212.727,A -85,B 0,C 180,E1 -6291.025,E2 -6291.025} C_VEL
LIN {X 0,Y 495.81,Z 212.728,A -85,B 0,C 180,E1 -6293.485,E2 -6293.485} C_VEL
LIN {X 0,Y 495.681,Z 212.739,A -85,B 0,C 180,E1 -6295.93,E2 -6295.93} C_VEL
LIN {X 0,Y 495.959,Z 212.71,A -85,B 0,C 180,E1 -6297.559,E2 -6297.559} C_VEL
LIN {X 0,Y 495.953,Z 212.704,A -85,B 0,C 180,E1 -6299.995,E2 -6299.995} C_VEL
LIN {X 0,Y 495.964,Z 212.7,A -85,B 0,C 180,E1 -6302.432,E2 -6302.432} C_VEL
LIN {X 0,Y 495.826,Z 212.723,A -85,B 0,C 180,E1 -6305.689,E2 -6305.689} C_VEL
LIN {X 0,Y 495.794,Z 212.723,A -85,B 0,C 180,E1 -6308.144,E2 -6308.144} C_VEL
LIN {X 0,Y 495.827,Z 212.727,A -85,B 0,C 180,E1 -6311.44,E2 -6311.44} C_VEL
LIN {X 0,Y 495.751,Z 212.728,A -85,B 0,C 180,E1 -6314.778,E2 -6314.778} C_VEL
LIN {X 0,Y 495.727,Z 212.737,A -85,B 0,C 180,E1 -6317.315,E2 -6317.315} C_VEL
LIN {X 0,Y 495.738,Z 212.731,A -85,B 0,C 180,E1 -6319.886,E2 -6319.886} C_VEL
LIN {X 0,Y 495.727,Z 212.732,A -85,B 0,C 180,E1 -6322.855,E2 -6322.855} C_VEL
LIN {X 0,Y 495.721,Z 212.732,A -85,B 0,C 180,E1 -6326.065,E2 -6326.065} C_VEL
LIN {X 0,Y 495.732,Z 212.731,A -85,B 0,C 180,E1 -6328.81,E2 -6328.81} C_VEL
LIN {X 0,Y 495.716,Z 212.735,A -85,B 0,C 180,E1 -6331.72,E2 -6331.72} C_VEL
LIN {X 0,Y 495.727,Z 212.731,A -85,B 0,C 180,E1 -6334.689,E2 -6334.689} C_VEL
LIN {X 0,Y 495.685,Z 212.74,A -85,B 0,C 180,E1 -6337.557,E2 -6337.557} C_VEL
LIN {X 0,Y 495.721,Z 212.732,A -85,B 0,C 180,E1 -6340.695,E2 -6340.695} C_VEL
LIN {X 0,Y 495.686,Z 212.736,A -85,B 0,C 180,E1 -6343.997,E2 -6343.997} C_VEL
LIN {X 0,Y 495.675,Z 212.743,A -85,B 0,C 180,E1 -6347.113,E2 -6347.113} C_VEL
LIN {X 0,Y 495.708,Z 212.733,A -85,B 0,C 180,E1 -6349.949,E2 -6349.949} C_VEL
LIN {X 0,Y 495.68,Z 212.737,A -85,B 0,C 180,E1 -6352.548,E2 -6352.548} C_VEL
LIN {X 0,Y 495.731,Z 212.735,A -85,B 0,C 180,E1 -6355.454,E2 -6355.454} C_VEL
LIN {X 0,Y 495.7,Z 212.733,A -85,B 0,C 180,E1 -6358.361,E2 -6358.361} C_VEL
LIN {X 0,Y 495.706,Z 212.735,A -85,B 0,C 180,E1 -6360.707,E2 -6360.707} C_VEL
LIN {X 0,Y 495.042,Z 212.823,A -85,B 0,C 180,E1 -6361.386,E2 -6361.386} C_VEL
LIN {X 0,Y 492.186,Z 213.176,A -85,B 0,C 180,E1 -6362.489,E2 -6362.489} C_VEL
LIN {X 0,Y 489.779,Z 213.477,A -85,B 0,C 180,E1 -6363.377,E2 -6363.377} C_VEL
LIN {X 0,Y 488.761,Z 213.598,A -85,B 0,C 180,E1 -6364.064,E2 -6364.064} C_VEL
LIN {X 0,Y 488.686,Z 213.607,A -85,B 0,C 180,E1 -6364.296,E2 -6364.296} C_VEL
LIN {X 0,Y 488.688,Z 213.616,A -85,B 0,C 180,E1 -6367.152,E2 -6367.152} C_VEL
LIN {X 0,Y 488.667,Z 213.61,A -85,B 0,C 180,E1 -6369.808,E2 -6369.808} C_VEL
LIN {X 0,Y 488.685,Z 213.608,A -85,B 0,C 180,E1 -6372.422,E2 -6372.422} C_VEL
LIN {X 0,Y 488.697,Z 213.613,A -85,B 0,C 180,E1 -6374.998,E2 -6374.998} C_VEL
LIN {X 0,Y 488.769,Z 213.597,A -85,B 0,C 180,E1 -6378.387,E2 -6378.387} C_VEL
LIN {X 0,Y 488.783,Z 213.596,A -85,B 0,C 180,E1 -6381.733,E2 -6381.733} C_VEL
LIN {X 0,Y 488.813,Z 213.591,A -85,B 0,C 180,E1 -6384.224,E2 -6384.224} C_VEL
LIN {X 0,Y 488.901,Z 213.583,A -85,B 0,C 180,E1 -6387.528,E2 -6387.528} C_VEL
LIN {X 0,Y 488.9,Z 213.58,A -85,B 0,C 180,E1 -6390,E2 -6390} C_VEL
LIN {X 0,Y 488.901,Z 213.582,A -85,B 0,C 180,E1 -6392.472,E2 -6392.472} C_VEL
LIN {X 0,Y 488.813,Z 213.592,A -85,B 0,C 180,E1 -6395.776,E2 -6395.776} C_VEL
LIN {X 0,Y 488.783,Z 213.597,A -85,B 0,C 180,E1 -6398.267,E2 -6398.267} C_VEL
LIN {X 0,Y 488.774,Z 213.603,A -85,B 0,C 180,E1 -6401.613,E2 -6401.613} C_VEL
LIN {X 0,Y 488.788,Z 213.695,A -85,B 0,C 180,E1 -6402.587,E2 -6402.587} C_VEL
LIN {X 0,Y 489.624,Z 220.046,A -85,B 0,C 180,E1 -6403.911,E2 -6403.911} C_VEL
LIN {X 0,Y 489.345,Z 232.785,A -85,B 0,C 180,E1 -6406.456,E2 -6406.456} C_VEL
LIN {X 0,Y 489.309,Z 234.522,A -85,B 0,C 180,E1 -6406.801,E2 -6406.801} C_VEL
LIN {X 0,Y 491.799,Z 247.846,A -85,B 0,C 180,E1 -6407.088,E2 -6407.088} C_VEL
LIN {X 0,Y 491.089,Z 341.384,A -85,B 0,C 180,E1 -6408.493,E2 -6408.493} C_VEL
LIN {X 0,Y 490.858,Z 354.633,A -85,B 0,C 180,E1 -6408.857,E2 -6408.857} C_VEL
LIN {X 0,Y 490.576,Z 366.66,A -85,B 0,C 180,E1 -6409.346,E2 -6409.346} C_VEL
LIN {X 0,Y 490.247,Z 378.796,A -85,B 0,C 180,E1 -6410.014,E2 -6410.014} C_VEL
LIN {X 0,Y 489.848,Z 389.803,A -85,B 0,C 180,E1 -6410.799,E2 -6410.799} C_VEL
LIN {X 0,Y 489.384,Z 401.152,A -85,B 0,C 180,E1 -6411.815,E2 -6411.815} C_VEL
LIN {X 0,Y 489.026,Z 410.258,A -85,B 0,C 180,E1 -6412.831,E2 -6412.831} C_VEL
LIN {X 0,Y 488.687,Z 418.57,A -85,B 0,C 180,E1 -6413.97,E2 -6413.97} C_VEL
LIN {X 0,Y 488.445,Z 426.119,A -85,B 0,C 180,E1 -6415.249,E2 -6415.249} C_VEL
LIN {X 0,Y 488.224,Z 432.045,A -85,B 0,C 180,E1 -6416.502,E2 -6416.502} C_VEL
LIN {X 0,Y 488.068,Z 437.185,A -85,B 0,C 180,E1 -6417.903,E2 -6417.903} C_VEL
LIN {X 0,Y 487.949,Z 440.972,A -85,B 0,C 180,E1 -6419.32,E2 -6419.32} C_VEL
LIN {X 0,Y 487.87,Z 442.821,A -85,B 0,C 180,E1 -6420.277,E2 -6420.277} C_VEL
LIN {X 0,Y 487.805,Z 444.615,A -85,B 0,C 180,E1 -6421.799,E2 -6421.799} C_VEL
LIN {X 0,Y 487.799,Z 445.034,A -85,B 0,C 180,E1 -6423.331,E2 -6423.331} C_VEL
LIN {X 0,Y 487.813,Z 444.17,A -85,B 0,C 180,E1 -6424.807,E2 -6424.807} C_VEL
LIN {X 0,Y 487.9,Z 442.109,A -85,B 0,C 180,E1 -6426.242,E2 -6426.242} C_VEL
LIN {X 0,Y 488.042,Z 438.887,A -85,B 0,C 180,E1 -6427.637,E2 -6427.637} C_VEL
LIN {X 0,Y 488.151,Z 434.519,A -85,B 0,C 180,E1 -6428.984,E2 -6428.984} C_VEL
LIN {X 0,Y 488.33,Z 428.64,A -85,B 0,C 180,E1 -6430.362,E2 -6430.362} C_VEL
LIN {X 0,Y 488.565,Z 422.017,A -85,B 0,C 180,E1 -6431.592,E2 -6431.592} C_VEL
LIN {X 0,Y 488.856,Z 414.754,A -85,B 0,C 180,E1 -6432.691,E2 -6432.691} C_VEL
LIN {X 0,Y 489.278,Z 405.285,A -85,B 0,C 180,E1 -6433.855,E2 -6433.855} C_VEL
LIN {X 0,Y 489.633,Z 395.118,A -85,B 0,C 180,E1 -6434.861,E2 -6434.861} C_VEL
LIN {X 0,Y 490.078,Z 384.195,A -85,B 0,C 180,E1 -6435.73,E2 -6435.73} C_VEL
LIN {X 0,Y 490.492,Z 372.125,A -85,B 0,C 180,E1 -6436.478,E2 -6436.478} C_VEL
LIN {X 0,Y 490.816,Z 359.688,A -85,B 0,C 180,E1 -6437.058,E2 -6437.058} C_VEL
LIN {X 0,Y 491.047,Z 346.769,A -85,B 0,C 180,E1 -6437.482,E2 -6437.482} C_VEL
LIN {X 0,Y 491.216,Z 332.541,A -85,B 0,C 180,E1 -6437.753,E2 -6437.753} C_VEL
LIN {X 0,Y 491.725,Z 246.577,A -85,B 0,C 180,E1 -6439.038,E2 -6439.038} C_VEL
LIN {X 0,Y 489.355,Z 234.36,A -85,B 0,C 180,E1 -6439.325,E2 -6439.325} C_VEL
LIN {X 0,Y 489.543,Z 219.216,A -85,B 0,C 180,E1 -6442.145,E2 -6442.145} C_VEL
LIN {X 0,Y 488.724,Z 213.611,A -85,B 0,C 180,E1 -6443.233,E2 -6443.233} C_VEL
LIN {X 0,Y 488.698,Z 213.611,A -85,B 0,C 180,E1 -6446.52,E2 -6446.52} C_VEL
LIN {X 0,Y 488.697,Z 213.609,A -85,B 0,C 180,E1 -6449.786,E2 -6449.786} C_VEL
LIN {X 0,Y 488.765,Z 213.606,A -85,B 0,C 180,E1 -6453.06,E2 -6453.06} C_VEL
LIN {X 0,Y 488.661,Z 213.612,A -85,B 0,C 180,E1 -6456.26,E2 -6456.26} C_VEL
LIN {X 0,Y 488.717,Z 213.61,A -85,B 0,C 180,E1 -6459.181,E2 -6459.181} C_VEL
LIN {X 0,Y 488.708,Z 213.609,A -85,B 0,C 180,E1 -6462.428,E2 -6462.428} C_VEL
LIN {X 0,Y 488.737,Z 213.607,A -85,B 0,C 180,E1 -6465.005,E2 -6465.005} C_VEL
LIN {X 0,Y 488.811,Z 213.594,A -85,B 0,C 180,E1 -6468.393,E2 -6468.393} C_VEL
LIN {X 0,Y 488.767,Z 213.596,A -85,B 0,C 180,E1 -6471.738,E2 -6471.738} C_VEL
LIN {X 0,Y 488.825,Z 213.592,A -85,B 0,C 180,E1 -6474.229,E2 -6474.229} C_VEL
LIN {X 0,Y 488.942,Z 213.575,A -85,B 0,C 180,E1 -6477.533,E2 -6477.533} C_VEL
LIN {X 0,Y 488.922,Z 213.584,A -85,B 0,C 180,E1 -6480.828,E2 -6480.828} C_VEL
LIN {X 0,Y 488.936,Z 213.579,A -85,B 0,C 180,E1 -6482.476,E2 -6482.476} C_VEL
LIN {X 0,Y 488.825,Z 213.587,A -85,B 0,C 180,E1 -6485.78,E2 -6485.78} C_VEL
LIN {X 0,Y 488.766,Z 213.6,A -85,B 0,C 180,E1 -6488.271,E2 -6488.271} C_VEL
LIN {X 0,Y 488.797,Z 213.594,A -85,B 0,C 180,E1 -6491.617,E2 -6491.617} C_VEL
LIN {X 0,Y 488.756,Z 213.602,A -85,B 0,C 180,E1 -6495.004,E2 -6495.004} C_VEL
LIN {X 0,Y 488.743,Z 213.605,A -85,B 0,C 180,E1 -6498.446,E2 -6498.446} C_VEL
LIN {X 0,Y 488.706,Z 213.607,A -85,B 0,C 180,E1 -6501.074,E2 -6501.074} C_VEL
LIN {X 0,Y 488.662,Z 213.61,A -85,B 0,C 180,E1 -6503.751,E2 -6503.751} C_VEL
LIN {X 0,Y 488.668,Z 213.614,A -85,B 0,C 180,E1 -6506.481,E2 -6506.481} C_VEL
LIN {X 0,Y 488.708,Z 213.604,A -85,B 0,C 180,E1 -6509.275,E2 -6509.275} C_VEL
LIN {X 0,Y 488.696,Z 213.611,A -85,B 0,C 180,E1 -6512.151,E2 -6512.151} C_VEL
LIN {X 0,Y 488.707,Z 213.606,A -85,B 0,C 180,E1 -6515.119,E2 -6515.119} C_VEL
LIN {X 0,Y 488.653,Z 213.617,A -85,B 0,C 180,E1 -6518.206,E2 -6518.206} C_VEL
LIN {X 0,Y 488.651,Z 213.614,A -85,B 0,C 180,E1 -6521.425,E2 -6521.425} C_VEL
LIN {X 0,Y 488.7,Z 213.611,A -85,B 0,C 180,E1 -6524.806,E2 -6524.806} C_VEL
LIN {X 0,Y 488.653,Z 213.614,A -85,B 0,C 180,E1 -6527.472,E2 -6527.472} C_VEL
LIN {X 0,Y 488.671,Z 213.613,A -85,B 0,C 180,E1 -6530.744,E2 -6530.744} C_VEL
LIN {X 0,Y 488.641,Z 213.618,A -85,B 0,C 180,E1 -6533.866,E2 -6533.866} C_VEL
LIN {X 0,Y 488.698,Z 213.613,A -85,B 0,C 180,E1 -6536.526,E2 -6536.526} C_VEL
LIN {X 0,Y 488.658,Z 213.617,A -85,B 0,C 180,E1 -6539.651,E2 -6539.651} C_VEL
LIN {X 0,Y 488.662,Z 213.617,A -85,B 0,C 180,E1 -6542.599,E2 -6542.599} C_VEL
LIN {X 0,Y 488.701,Z 213.725,A -85,B 0,C 180,E1 -6544.719,E2 -6544.719} C_VEL
LIN {X 0,Y 490.528,Z 223.701,A -85,B 0,C 180,E1 -6546.488,E2 -6546.488} C_VEL
LIN {X 0,Y 490.109,Z 238.852,A -85,B 0,C 180,E1 -6548.993,E2 -6548.993} C_VEL
LIN {X 0,Y 489.492,Z 258.743,A -85,B 0,C 180,E1 -6552.236,E2 -6552.236} C_VEL
LIN {X 0,Y 489.248,Z 267.962,A -85,B 0,C 180,E1 -6553.723,E2 -6553.723} C_VEL
LIN {X 0,Y 491.635,Z 285.056,A -85,B 0,C 180,E1 -6554.065,E2 -6554.065} C_VEL
LIN {X 0,Y 491.072,Z 376.505,A -85,B 0,C 180,E1 -6555.443,E2 -6555.443} C_VEL
LIN {X 0,Y 490.717,Z 389.738,A -85,B 0,C 180,E1 -6555.803,E2 -6555.803} C_VEL
LIN {X 0,Y 490.355,Z 402.47,A -85,B 0,C 180,E1 -6556.321,E2 -6556.321} C_VEL
LIN {X 0,Y 489.975,Z 413.802,A -85,B 0,C 180,E1 -6556.944,E2 -6556.944} C_VEL
LIN {X 0,Y 489.519,Z 425.501,A -85,B 0,C 180,E1 -6557.775,E2 -6557.775} C_VEL
LIN {X 0,Y 489.138,Z 436.034,A -85,B 0,C 180,E1 -6558.711,E2 -6558.711} C_VEL
LIN {X 0,Y 488.793,Z 444.649,A -85,B 0,C 180,E1 -6559.646,E2 -6559.646} C_VEL
LIN {X 0,Y 488.485,Z 452.598,A -85,B 0,C 180,E1 -6560.686,E2 -6560.686} C_VEL
LIN {X 0,Y 488.257,Z 460.366,A -85,B 0,C 180,E1 -6561.933,E2 -6561.933} C_VEL
LIN {X 0,Y 488.097,Z 465.683,A -85,B 0,C 180,E1 -6562.97,E2 -6562.97} C_VEL
LIN {X 0,Y 488.014,Z 470.841,A -85,B 0,C 180,E1 -6564.214,E2 -6564.214} C_VEL
LIN {X 0,Y 487.921,Z 474.844,A -85,B 0,C 180,E1 -6565.456,E2 -6565.456} C_VEL
LIN {X 0,Y 487.967,Z 477.806,A -85,B 0,C 180,E1 -6566.697,E2 -6566.697} C_VEL
LIN {X 0,Y 487.912,Z 479.215,A -85,B 0,C 180,E1 -6567.523,E2 -6567.523} C_VEL
LIN {X 0,Y 487.894,Z 480.222,A -85,B 0,C 180,E1 -6568.349,E2 -6568.349} C_VEL
LIN {X 0,Y 487.826,Z 481.06,A -85,B 0,C 180,E1 -6570,E2 -6570} C_VEL
LIN {X 0,Y 487.894,Z 480.243,A -85,B 0,C 180,E1 -6571.651,E2 -6571.651} C_VEL
LIN {X 0,Y 487.912,Z 479.246,A -85,B 0,C 180,E1 -6572.477,E2 -6572.477} C_VEL
LIN {X 0,Y 487.967,Z 477.847,A -85,B 0,C 180,E1 -6573.303,E2 -6573.303} C_VEL
LIN {X 0,Y 487.921,Z 474.897,A -85,B 0,C 180,E1 -6574.544,E2 -6574.544} C_VEL
LIN {X 0,Y 488.014,Z 470.905,A -85,B 0,C 180,E1 -6575.786,E2 -6575.786} C_VEL
LIN {X 0,Y 488.139,Z 464.758,A -85,B 0,C 180,E1 -6577.237,E2 -6577.237} C_VEL
LIN {X 0,Y 488.359,Z 458.046,A -85,B 0,C 180,E1 -6578.482,E2 -6578.482} C_VEL
LIN {X 0,Y 488.653,Z 449.717,A -85,B 0,C 180,E1 -6579.729,E2 -6579.729} C_VEL
LIN {X 0,Y 488.971,Z 441.163,A -85,B 0,C 180,E1 -6580.769,E2 -6580.769} C_VEL
LIN {X 0,Y 489.427,Z 430.602,A -85,B 0,C 180,E1 -6581.807,E2 -6581.807} C_VEL
LIN {X 0,Y 489.768,Z 419.002,A -85,B 0,C 180,E1 -6582.724,E2 -6582.724} C_VEL
LIN {X 0,Y 490.203,Z 406.685,A -85,B 0,C 180,E1 -6583.472,E2 -6583.472} C_VEL
LIN {X 0,Y 490.601,Z 394.178,A -85,B 0,C 180,E1 -6584.042,E2 -6584.042} C_VEL
LIN {X 0,Y 490.923,Z 381.139,A -85,B 0,C 180,E1 -6584.455,E2 -6584.455} C_VEL
LIN {X 0,Y 491.156,Z 365.45,A -85,B 0,C 180,E1 -6584.74,E2 -6584.74} C_VEL
LIN {X 0,Y 491.481,Z 282.938,A -85,B 0,C 180,E1 -6585.971,E2 -6585.971} C_VEL
LIN {X 0,Y 489.263,Z 268.323,A -85,B 0,C 180,E1 -6586.269,E2 -6586.269} C_VEL
LIN {X 0,Y 489.876,Z 248.778,A -85,B 0,C 180,E1 -6589.484,E2 -6589.484} C_VEL
LIN {X 0,Y 490.483,Z 231.807,A -85,B 0,C 180,E1 -6592.315,E2 -6592.315} C_VEL
LIN {X 0,Y 490.665,Z 223.964,A -85,B 0,C 180,E1 -6593.644,E2 -6593.644} C_VEL
LIN {X 0,Y 488.706,Z 213.612,A -85,B 0,C 180,E1 -6595.557,E2 -6595.557} C_VEL
LIN {X 0,Y 488.66,Z 213.614,A -85,B 0,C 180,E1 -6598.677,E2 -6598.677} C_VEL
LIN {X 0,Y 488.684,Z 213.614,A -85,B 0,C 180,E1 -6601.947,E2 -6601.947} C_VEL
LIN {X 0,Y 488.659,Z 213.611,A -85,B 0,C 180,E1 -6605.119,E2 -6605.119} C_VEL
LIN {X 0,Y 488.646,Z 213.615,A -85,B 0,C 180,E1 -6608.202,E2 -6608.202} C_VEL
LIN {X 0,Y 488.669,Z 213.611,A -85,B 0,C 180,E1 -6610.335,E2 -6610.335} C_VEL
LIN {X 0,Y 488.631,Z 213.621,A -85,B 0,C 180,E1 -6613.659,E2 -6613.659} C_VEL
LIN {X 0,Y 488.666,Z 213.611,A -85,B 0,C 180,E1 -6616.34,E2 -6616.34} C_VEL
LIN {X 0,Y 488.672,Z 213.617,A -85,B 0,C 180,E1 -6619.667,E2 -6619.667} C_VEL
LIN {X 0,Y 488.625,Z 213.615,A -85,B 0,C 180,E1 -6622.833,E2 -6622.833} C_VEL
LIN {X 0,Y 488.701,Z 213.611,A -85,B 0,C 180,E1 -6625.882,E2 -6625.882} C_VEL
LIN {X 0,Y 488.659,Z 213.611,A -85,B 0,C 180,E1 -6628.815,E2 -6628.815} C_VEL
LIN {X 0,Y 488.675,Z 213.617,A -85,B 0,C 180,E1 -6631.663,E2 -6631.663} C_VEL
LIN {X 0,Y 488.691,Z 213.607,A -85,B 0,C 180,E1 -6634.958,E2 -6634.958} C_VEL
LIN {X 0,Y 488.688,Z 213.61,A -85,B 0,C 180,E1 -6638.039,E2 -6638.039} C_VEL
LIN {X 0,Y 488.704,Z 213.605,A -85,B 0,C 180,E1 -6640.681,E2 -6640.681} C_VEL
LIN {X 0,Y 488.748,Z 213.601,A -85,B 0,C 180,E1 -6644.141,E2 -6644.141} C_VEL
LIN {X 0,Y 488.725,Z 213.611,A -85,B 0,C 180,E1 -6647.539,E2 -6647.539} C_VEL
LIN {X 0,Y 488.717,Z 213.604,A -85,B 0,C 180,E1 -6650.894,E2 -6650.894} C_VEL
LIN {X 0,Y 488.764,Z 213.604,A -85,B 0,C 180,E1 -6653.39,E2 -6653.39} C_VEL
LIN {X 0,Y 488.642,Z 213.616,A -85,B 0,C 180,E1 -6655.872,E2 -6655.872} C_VEL
LIN {X 0,Y 488.926,Z 213.586,A -85,B 0,C 180,E1 -6657.524,E2 -6657.524} C_VEL
LIN {X 0,Y 488.923,Z 213.58,A -85,B 0,C 180,E1 -6659.995,E2 -6659.995} C_VEL
LIN {X 0,Y 488.931,Z 213.576,A -85,B 0,C 180,E1 -6662.467,E2 -6662.467} C_VEL
LIN {X 0,Y 488.786,Z 213.599,A -85,B 0,C 180,E1 -6665.772,E2 -6665.772} C_VEL
LIN {X 0,Y 488.741,Z 213.601,A -85,B 0,C 180,E1 -6668.262,E2 -6668.262} C_VEL
LIN {X 0,Y 488.782,Z 213.602,A -85,B 0,C 180,E1 -6671.608,E2 -6671.608} C_VEL
LIN {X 0,Y 488.728,Z 213.605,A -85,B 0,C 180,E1 -6674.996,E2 -6674.996} C_VEL
LIN {X 0,Y 488.719,Z 213.603,A -85,B 0,C 180,E1 -6678.437,E2 -6678.437} C_VEL
LIN {X 0,Y 488.677,Z 213.612,A -85,B 0,C 180,E1 -6681.066,E2 -6681.066} C_VEL
LIN {X 0,Y 488.638,Z 213.617,A -85,B 0,C 180,E1 -6683.742,E2 -6683.742} C_VEL
LIN {X 0,Y 488.713,Z 213.607,A -85,B 0,C 180,E1 -6686.928,E2 -6686.928} C_VEL
LIN {X 0,Y 488.685,Z 213.615,A -85,B 0,C 180,E1 -6689.266,E2 -6689.266} C_VEL
LIN {X 0,Y 488.664,Z 213.61,A -85,B 0,C 180,E1 -6692.142,E2 -6692.142} C_VEL
LIN {X 0,Y 488.675,Z 213.614,A -85,B 0,C 180,E1 -6695.11,E2 -6695.11} C_VEL
LIN {X 0,Y 488.635,Z 213.613,A -85,B 0,C 180,E1 -6698.196,E2 -6698.196} C_VEL
LIN {X 0,Y 488.673,Z 213.609,A -85,B 0,C 180,E1 -6700.34,E2 -6700.34} C_VEL
LIN {X 0,Y 488.639,Z 213.616,A -85,B 0,C 180,E1 -6703.65,E2 -6703.65} C_VEL
LIN {X 0,Y 488.637,Z 213.613,A -85,B 0,C 180,E1 -6706.341,E2 -6706.341} C_VEL
LIN {X 0,Y 488.681,Z 213.611,A -85,B 0,C 180,E1 -6709.673,E2 -6709.673} C_VEL
LIN {X 0,Y 488.632,Z 213.617,A -85,B 0,C 180,E1 -6712.838,E2 -6712.838} C_VEL
LIN {X 0,Y 488.68,Z 213.609,A -85,B 0,C 180,E1 -6715.884,E2 -6715.884} C_VEL
LIN {X 0,Y 488.638,Z 213.616,A -85,B 0,C 180,E1 -6718.817,E2 -6718.817} C_VEL
LIN {X 0,Y 488.687,Z 213.609,A -85,B 0,C 180,E1 -6721.668,E2 -6721.668} C_VEL
LIN {X 0,Y 488.686,Z 213.607,A -85,B 0,C 180,E1 -6724.296,E2 -6724.296} C_VEL
LIN {X 0,Y 488.038,Z 213.695,A -85,B 0,C 180,E1 -6724.984,E2 -6724.984} C_VEL
LIN {X 0,Y 485.179,Z 214.048,A -85,B 0,C 180,E1 -6726.101,E2 -6726.101} C_VEL
LIN {X 0,Y 482.744,Z 214.354,A -85,B 0,C 180,E1 -6727,E2 -6727} C_VEL
LIN {X 0,Y 481.692,Z 214.481,A -85,B 0,C 180,E1 -6727.696,E2 -6727.696} C_VEL
LIN {X 0,Y 481.603,Z 214.49,A -85,B 0,C 180,E1 -6727.931,E2 -6727.931} C_VEL
LIN {X 0,Y 481.646,Z 214.485,A -85,B 0,C 180,E1 -6730.391,E2 -6730.391} C_VEL
LIN {X 0,Y 481.638,Z 214.492,A -85,B 0,C 180,E1 -6733.032,E2 -6733.032} C_VEL
LIN {X 0,Y 481.627,Z 214.488,A -85,B 0,C 180,E1 -6735.637,E2 -6735.637} C_VEL
LIN {X 0,Y 481.732,Z 214.473,A -85,B 0,C 180,E1 -6738.215,E2 -6738.215} C_VEL
LIN {X 0,Y 481.725,Z 214.476,A -85,B 0,C 180,E1 -6741.611,E2 -6741.611} C_VEL
LIN {X 0,Y 481.773,Z 214.468,A -85,B 0,C 180,E1 -6744.139,E2 -6744.139} C_VEL
LIN {X 0,Y 481.869,Z 214.459,A -85,B 0,C 180,E1 -6747.492,E2 -6747.492} C_VEL
LIN {X 0,Y 481.871,Z 214.456,A -85,B 0,C 180,E1 -6750,E2 -6750} C_VEL
LIN {X 0,Y 481.869,Z 214.458,A -85,B 0,C 180,E1 -6752.508,E2 -6752.508} C_VEL
LIN {X 0,Y 481.773,Z 214.468,A -85,B 0,C 180,E1 -6755.861,E2 -6755.861} C_VEL
LIN {X 0,Y 481.725,Z 214.477,A -85,B 0,C 180,E1 -6758.389,E2 -6758.389} C_VEL
LIN {X 0,Y 481.749,Z 214.478,A -85,B 0,C 180,E1 -6762.234,E2 -6762.234} C_VEL
LIN {X 0,Y 481.742,Z 214.51,A -85,B 0,C 180,E1 -6762.42,E2 -6762.42} C_VEL
LIN {X 0,Y 482.668,Z 221.539,A -85,B 0,C 180,E1 -6763.901,E2 -6763.901} C_VEL
LIN {X 0,Y 482.342,Z 234.691,A -85,B 0,C 180,E1 -6766.551,E2 -6766.551} C_VEL
LIN {X 0,Y 484.974,Z 248.782,A -85,B 0,C 180,E1 -6766.871,E2 -6766.871} C_VEL
LIN {X 0,Y 484.212,Z 341.847,A -85,B 0,C 180,E1 -6768.292,E2 -6768.292} C_VEL
LIN {X 0,Y 483.962,Z 355.771,A -85,B 0,C 180,E1 -6768.688,E2 -6768.688} C_VEL
LIN {X 0,Y 483.662,Z 367.951,A -85,B 0,C 180,E1 -6769.202,E2 -6769.202} C_VEL
LIN {X 0,Y 483.315,Z 379.642,A -85,B 0,C 180,E1 -6769.87,E2 -6769.87} C_VEL
LIN {X 0,Y 482.881,Z 390.558,A -85,B 0,C 180,E1 -6770.667,E2 -6770.667} C_VEL
LIN {X 0,Y 482.433,Z 400.656,A -85,B 0,C 180,E1 -6771.582,E2 -6771.582} C_VEL
LIN {X 0,Y 482.092,Z 408.965,A -85,B 0,C 180,E1 -6772.499,E2 -6772.499} C_VEL
LIN {X 0,Y 481.752,Z 417.587,A -85,B 0,C 180,E1 -6773.651,E2 -6773.651} C_VEL
LIN {X 0,Y 481.396,Z 425.898,A -85,B 0,C 180,E1 -6775.047,E2 -6775.047} C_VEL
LIN {X 0,Y 481.154,Z 432.496,A -85,B 0,C 180,E1 -6776.455,E2 -6776.455} C_VEL
LIN {X 0,Y 480.99,Z 437.577,A -85,B 0,C 180,E1 -6777.876,E2 -6777.876} C_VEL
LIN {X 0,Y 480.872,Z 441.328,A -85,B 0,C 180,E1 -6779.314,E2 -6779.314} C_VEL
LIN {X 0,Y 480.736,Z 443.848,A -85,B 0,C 180,E1 -6780.774,E2 -6780.774} C_VEL
LIN {X 0,Y 480.719,Z 445.016,A -85,B 0,C 180,E1 -6782.026,E2 -6782.026} C_VEL
LIN {X 0,Y 480.697,Z 445.208,A -85,B 0,C 180,E1 -6783.749,E2 -6783.749} C_VEL
LIN {X 0,Y 480.742,Z 444.212,A -85,B 0,C 180,E1 -6785.062,E2 -6785.062} C_VEL
LIN {X 0,Y 480.831,Z 441.953,A -85,B 0,C 180,E1 -6786.508,E2 -6786.508} C_VEL
LIN {X 0,Y 480.977,Z 438.54,A -85,B 0,C 180,E1 -6787.916,E2 -6787.916} C_VEL
LIN {X 0,Y 481.117,Z 433.997,A -85,B 0,C 180,E1 -6789.279,E2 -6789.279} C_VEL
LIN {X 0,Y 481.302,Z 428.251,A -85,B 0,C 180,E1 -6790.608,E2 -6790.608} C_VEL
LIN {X 0,Y 481.611,Z 421.103,A -85,B 0,C 180,E1 -6791.918,E2 -6791.918} C_VEL
LIN {X 0,Y 481.931,Z 414.134,A -85,B 0,C 180,E1 -6792.957,E2 -6792.957} C_VEL
LIN {X 0,Y 482.331,Z 404.881,A -85,B 0,C 180,E1 -6794.086,E2 -6794.086} C_VEL
LIN {X 0,Y 482.72,Z 394.904,A -85,B 0,C 180,E1 -6795.077,E2 -6795.077} C_VEL
LIN {X 0,Y 483.201,Z 383.26,A -85,B 0,C 180,E1 -6796,E2 -6796} C_VEL
LIN {X 0,Y 483.626,Z 371.284,A -85,B 0,C 180,E1 -6796.733,E2 -6796.733} C_VEL
LIN {X 0,Y 483.99,Z 359.068,A -85,B 0,C 180,E1 -6797.296,E2 -6797.296} C_VEL
LIN {X 0,Y 484.207,Z 347.074,A -85,B 0,C 180,E1 -6797.689,E2 -6797.689} C_VEL
LIN {X 0,Y 484.373,Z 332.65,A -85,B 0,C 180,E1 -6797.969,E2 -6797.969} C_VEL
LIN {X 0,Y 484.901,Z 247.326,A -85,B 0,C 180,E1 -6799.266,E2 -6799.266} C_VEL
LIN {X 0,Y 482.4,Z 234.647,A -85,B 0,C 180,E1 -6799.564,E2 -6799.564} C_VEL
LIN {X 0,Y 482.556,Z 220.082,A -85,B 0,C 180,E1 -6802.297,E2 -6802.297} C_VEL
LIN {X 0,Y 481.677,Z 214.488,A -85,B 0,C 180,E1 -6803.438,E2 -6803.438} C_VEL
LIN {X 0,Y 481.67,Z 214.486,A -85,B 0,C 180,E1 -6806.335,E2 -6806.335} C_VEL
LIN {X 0,Y 481.622,Z 214.494,A -85,B 0,C 180,E1 -6809.421,E2 -6809.421} C_VEL
LIN {X 0,Y 481.668,Z 214.483,A -85,B 0,C 180,E1 -6812.173,E2 -6812.173} C_VEL
LIN {X 0,Y 481.686,Z 214.488,A -85,B 0,C 180,E1 -6814.975,E2 -6814.975} C_VEL
LIN {X 0,Y 481.62,Z 214.489,A -85,B 0,C 180,E1 -6817.71,E2 -6817.71} C_VEL
LIN {X 0,Y 481.678,Z 214.484,A -85,B 0,C 180,E1 -6820.398,E2 -6820.398} C_VEL
LIN {X 0,Y 481.665,Z 214.49,A -85,B 0,C 180,E1 -6823.039,E2 -6823.039} C_VEL
LIN {X 0,Y 481.665,Z 214.483,A -85,B 0,C 180,E1 -6825.644,E2 -6825.644} C_VEL
LIN {X 0,Y 481.776,Z 214.469,A -85,B 0,C 180,E1 -6828.221,E2 -6828.221} C_VEL
LIN {X 0,Y 481.722,Z 214.474,A -85,B 0,C 180,E1 -6831.616,E2 -6831.616} C_VEL
LIN {X 0,Y 481.786,Z 214.468,A -85,B 0,C 180,E1 -6834.144,E2 -6834.144} C_VEL
LIN {X 0,Y 481.909,Z 214.451,A -85,B 0,C 180,E1 -6837.497,E2 -6837.497} C_VEL
LIN {X 0,Y 481.873,Z 214.462,A -85,B 0,C 180,E1 -6840.84,E2 -6840.84} C_VEL
LIN {X 0,Y 481.903,Z 214.455,A -85,B 0,C 180,E1 -6842.512,E2 -6842.512} C_VEL
LIN {X 0,Y 481.786,Z 214.464,A -85,B 0,C 180,E1 -6845.865,E2 -6845.865} C_VEL
LIN {X 0,Y 481.721,Z 214.48,A -85,B 0,C 180,E1 -6848.393,E2 -6848.393} C_VEL
LIN {X 0,Y 481.744,Z 214.473,A -85,B 0,C 180,E1 -6851.789,E2 -6851.789} C_VEL
LIN {X 0,Y 481.738,Z 214.474,A -85,B 0,C 180,E1 -6855.228,E2 -6855.228} C_VEL
LIN {X 0,Y 481.705,Z 214.481,A -85,B 0,C 180,E1 -6858.726,E2 -6858.726} C_VEL
LIN {X 0,Y 481.644,Z 214.484,A -85,B 0,C 180,E1 -6861.399,E2 -6861.399} C_VEL
LIN {X 0,Y 481.641,Z 214.487,A -85,B 0,C 180,E1 -6864.119,E2 -6864.119} C_VEL
LIN {X 0,Y 481.644,Z 214.485,A -85,B 0,C 180,E1 -6867.118,E2 -6867.118} C_VEL
LIN {X 0,Y 481.669,Z 214.481,A -85,B 0,C 180,E1 -6869.745,E2 -6869.745} C_VEL
LIN {X 0,Y 481.653,Z 214.487,A -85,B 0,C 180,E1 -6872.679,E2 -6872.679} C_VEL
LIN {X 0,Y 481.651,Z 214.485,A -85,B 0,C 180,E1 -6875.204,E2 -6875.204} C_VEL
LIN {X 0,Y 481.629,Z 214.49,A -85,B 0,C 180,E1 -6878.005,E2 -6878.005} C_VEL
LIN {X 0,Y 481.61,Z 214.492,A -85,B 0,C 180,E1 -6881.05,E2 -6881.05} C_VEL
LIN {X 0,Y 481.655,Z 214.491,A -85,B 0,C 180,E1 -6884.461,E2 -6884.461} C_VEL
LIN {X 0,Y 481.613,Z 214.493,A -85,B 0,C 180,E1 -6887.837,E2 -6887.837} C_VEL
LIN {X 0,Y 481.634,Z 214.491,A -85,B 0,C 180,E1 -6890.661,E2 -6890.661} C_VEL
LIN {X 0,Y 481.606,Z 214.491,A -85,B 0,C 180,E1 -6893.383,E2 -6893.383} C_VEL
LIN {X 0,Y 481.662,Z 214.491,A -85,B 0,C 180,E1 -6896.327,E2 -6896.327} C_VEL
LIN {X 0,Y 481.618,Z 214.493,A -85,B 0,C 180,E1 -6899.428,E2 -6899.428} C_VEL
LIN {X 0,Y 481.635,Z 214.494,A -85,B 0,C 180,E1 -6902.165,E2 -6902.165} C_VEL
LIN {X 0,Y 481.642,Z 214.593,A -85,B 0,C 180,E1 -6904.52,E2 -6904.52} C_VEL
LIN {X 0,Y 483.55,Z 224.448,A -85,B 0,C 180,E1 -6906.302,E2 -6906.302} C_VEL
LIN {X 0,Y 483.134,Z 239.907,A -85,B 0,C 180,E1 -6908.899,E2 -6908.899} C_VEL
LIN {X 0,Y 482.54,Z 258.476,A -85,B 0,C 180,E1 -6911.972,E2 -6911.972} C_VEL
LIN {X 0,Y 482.245,Z 267.63,A -85,B 0,C 180,E1 -6913.474,E2 -6913.474} C_VEL
LIN {X 0,Y 484.804,Z 286.022,A -85,B 0,C 180,E1 -6913.849,E2 -6913.849} C_VEL
LIN {X 0,Y 484.216,Z 376.214,A -85,B 0,C 180,E1 -6915.232,E2 -6915.232} C_VEL
LIN {X 0,Y 483.836,Z 389.445,A -85,B 0,C 180,E1 -6915.597,E2 -6915.597} C_VEL
LIN {X 0,Y 483.451,Z 402.181,A -85,B 0,C 180,E1 -6916.122,E2 -6916.122} C_VEL
LIN {X 0,Y 483.033,Z 413.517,A -85,B 0,C 180,E1 -6916.753,E2 -6916.753} C_VEL
LIN {X 0,Y 482.574,Z 425.249,A -85,B 0,C 180,E1 -6917.598,E2 -6917.598} C_VEL
LIN {X 0,Y 482.159,Z 435.756,A -85,B 0,C 180,E1 -6918.545,E2 -6918.545} C_VEL
LIN {X 0,Y 481.757,Z 444.37,A -85,B 0,C 180,E1 -6919.493,E2 -6919.493} C_VEL
LIN {X 0,Y 481.45,Z 452.321,A -85,B 0,C 180,E1 -6920.548,E2 -6920.548} C_VEL
LIN {X 0,Y 481.186,Z 460.09,A -85,B 0,C 180,E1 -6921.813,E2 -6921.813} C_VEL
LIN {X 0,Y 481.025,Z 465.41,A -85,B 0,C 180,E1 -6922.866,E2 -6922.866} C_VEL
LIN {X 0,Y 480.919,Z 470.569,A -85,B 0,C 180,E1 -6924.129,E2 -6924.129} C_VEL
LIN {X 0,Y 480.84,Z 474.576,A -85,B 0,C 180,E1 -6925.389,E2 -6925.389} C_VEL
LIN {X 0,Y 480.891,Z 477.541,A -85,B 0,C 180,E1 -6926.649,E2 -6926.649} C_VEL
LIN {X 0,Y 480.824,Z 479.96,A -85,B 0,C 180,E1 -6928.325,E2 -6928.325} C_VEL
LIN {X 0,Y 480.75,Z 480.799,A -85,B 0,C 180,E1 -6930,E2 -6930} C_VEL
LIN {X 0,Y 480.824,Z 479.982,A -85,B 0,C 180,E1 -6931.675,E2 -6931.675} C_VEL
LIN {X 0,Y 480.891,Z 477.584,A -85,B 0,C 180,E1 -6933.351,E2 -6933.351} C_VEL
LIN {X 0,Y 480.84,Z 474.632,A -85,B 0,C 180,E1 -6934.611,E2 -6934.611} C_VEL
LIN {X 0,Y 480.919,Z 470.637,A -85,B 0,C 180,E1 -6935.871,E2 -6935.871} C_VEL
LIN {X 0,Y 481.091,Z 464.487,A -85,B 0,C 180,E1 -6937.344,E2 -6937.344} C_VEL
LIN {X 0,Y 481.311,Z 457.769,A -85,B 0,C 180,E1 -6938.608,E2 -6938.608} C_VEL
LIN {X 0,Y 481.591,Z 449.432,A -85,B 0,C 180,E1 -6939.873,E2 -6939.873} C_VEL
LIN {X 0,Y 481.965,Z 440.868,A -85,B 0,C 180,E1 -6940.927,E2 -6940.927} C_VEL
LIN {X 0,Y 482.441,Z 430.37,A -85,B 0,C 180,E1 -6941.974,E2 -6941.974} C_VEL
LIN {X 0,Y 482.76,Z 420.107,A -85,B 0,C 180,E1 -6942.805,E2 -6942.805} C_VEL
LIN {X 0,Y 483.226,Z 408.308,A -85,B 0,C 180,E1 -6943.563,E2 -6943.563} C_VEL
LIN {X 0,Y 483.618,Z 396.389,A -85,B 0,C 180,E1 -6944.141,E2 -6944.141} C_VEL
LIN {X 0,Y 483.992,Z 382.631,A -85,B 0,C 180,E1 -6944.613,E2 -6944.613} C_VEL
LIN {X 0,Y 484.273,Z 370.138,A -85,B 0,C 180,E1 -6944.873,E2 -6944.873} C_VEL
LIN {X 0,Y 484.739,Z 284.452,A -85,B 0,C 180,E1 -6946.168,E2 -6946.168} C_VEL
LIN {X 0,Y 482.261,Z 268.066,A -85,B 0,C 180,E1 -6946.51,E2 -6946.51} C_VEL
LIN {X 0,Y 482.882,Z 249.822,A -85,B 0,C 180,E1 -6949.557,E2 -6949.557} C_VEL
LIN {X 0,Y 483.553,Z 232.854,A -85,B 0,C 180,E1 -6952.427,E2 -6952.427} C_VEL
LIN {X 0,Y 483.722,Z 225.193,A -85,B 0,C 180,E1 -6953.744,E2 -6953.744} C_VEL
LIN {X 0,Y 481.657,Z 214.491,A -85,B 0,C 180,E1 -6955.725,E2 -6955.725} C_VEL
LIN {X 0,Y 481.61,Z 214.492,A -85,B 0,C 180,E1 -6958.885,E2 -6958.885} C_VEL
LIN {X 0,Y 481.63,Z 214.49,A -85,B 0,C 180,E1 -6962.181,E2 -6962.181} C_VEL
LIN {X 0,Y 481.606,Z 214.49,A -85,B 0,C 180,E1 -6965.191,E2 -6965.191} C_VEL
LIN {X 0,Y 481.622,Z 214.493,A -85,B 0,C 180,E1 -6967.999,E2 -6967.999} C_VEL
LIN {X 0,Y 481.608,Z 214.489,A -85,B 0,C 180,E1 -6971.045,E2 -6971.045} C_VEL
LIN {X 0,Y 481.61,Z 214.489,A -85,B 0,C 180,E1 -6974.462,E2 -6974.462} C_VEL
LIN {X 0,Y 481.616,Z 214.488,A -85,B 0,C 180,E1 -6976.854,E2 -6976.854} C_VEL
LIN {X 0,Y 481.631,Z 214.49,A -85,B 0,C 180,E1 -6980.052,E2 -6980.052} C_VEL
LIN {X 0,Y 481.587,Z 214.494,A -85,B 0,C 180,E1 -6983.246,E2 -6983.246} C_VEL
LIN {X 0,Y 481.658,Z 214.484,A -85,B 0,C 180,E1 -6986.323,E2 -6986.323} C_VEL
LIN {X 0,Y 481.612,Z 214.493,A -85,B 0,C 180,E1 -6989.423,E2 -6989.423} C_VEL
LIN {X 0,Y 481.629,Z 214.488,A -85,B 0,C 180,E1 -6992.16,E2 -6992.16} C_VEL
LIN {X 0,Y 481.665,Z 214.483,A -85,B 0,C 180,E1 -6994.963,E2 -6994.963} C_VEL
LIN {X 0,Y 481.642,Z 214.492,A -85,B 0,C 180,E1 -6997.701,E2 -6997.701} C_VEL
LIN {X 0,Y 481.651,Z 214.484,A -85,B 0,C 180,E1 -7000.387,E2 -7000.387} C_VEL
LIN {X 0,Y 481.644,Z 214.486,A -85,B 0,C 180,E1 -7003.028,E2 -7003.028} C_VEL
LIN {X 0,Y 481.666,Z 214.49,A -85,B 0,C 180,E1 -7005.634,E2 -7005.634} C_VEL
LIN {X 0,Y 481.708,Z 214.478,A -85,B 0,C 180,E1 -7008.21,E2 -7008.21} C_VEL
LIN {X 0,Y 481.703,Z 214.485,A -85,B 0,C 180,E1 -7011.606,E2 -7011.606} C_VEL
LIN {X 0,Y 481.764,Z 214.471,A -85,B 0,C 180,E1 -7014.135,E2 -7014.135} C_VEL
LIN {X 0,Y 481.891,Z 214.462,A -85,B 0,C 180,E1 -7017.488,E2 -7017.488} C_VEL
LIN {X 0,Y 481.893,Z 214.456,A -85,B 0,C 180,E1 -7019.995,E2 -7019.995} C_VEL
LIN {X 0,Y 481.898,Z 214.453,A -85,B 0,C 180,E1 -7022.503,E2 -7022.503} C_VEL
LIN {X 0,Y 481.747,Z 214.475,A -85,B 0,C 180,E1 -7025.856,E2 -7025.856} C_VEL
LIN {X 0,Y 481.699,Z 214.477,A -85,B 0,C 180,E1 -7028.384,E2 -7028.384} C_VEL
LIN {X 0,Y 481.728,Z 214.478,A -85,B 0,C 180,E1 -7031.78,E2 -7031.78} C_VEL
LIN {X 0,Y 481.713,Z 214.481,A -85,B 0,C 180,E1 -7035.219,E2 -7035.219} C_VEL
LIN {X 0,Y 481.68,Z 214.481,A -85,B 0,C 180,E1 -7038.717,E2 -7038.717} C_VEL
LIN {X 0,Y 481.616,Z 214.497,A -85,B 0,C 180,E1 -7041.39,E2 -7041.39} C_VEL
LIN {X 0,Y 481.616,Z 214.488,A -85,B 0,C 180,E1 -7044.11,E2 -7044.11} C_VEL
LIN {X 0,Y 481.68,Z 214.485,A -85,B 0,C 180,E1 -7047.126,E2 -7047.126} C_VEL
LIN {X 0,Y 481.641,Z 214.488,A -85,B 0,C 180,E1 -7049.736,E2 -7049.736} C_VEL
LIN {X 0,Y 481.633,Z 214.487,A -85,B 0,C 180,E1 -7052.669,E2 -7052.669} C_VEL
LIN {X 0,Y 481.594,Z 214.494,A -85,B 0,C 180,E1 -7055.705,E2 -7055.705} C_VEL
LIN {X 0,Y 481.626,Z 214.489,A -85,B 0,C 180,E1 -7058.855,E2 -7058.855} C_VEL
LIN {X 0,Y 481.606,Z 214.49,A -85,B 0,C 180,E1 -7061.908,E2 -7061.908} C_VEL
LIN {X 0,Y 481.611,Z 214.489,A -85,B 0,C 180,E1 -7064.453,E2 -7064.453} C_VEL
LIN {X 0,Y 481.597,Z 214.492,A -85,B 0,C 180,E1 -7067.835,E2 -7067.835} C_VEL
LIN {X 0,Y 481.628,Z 214.488,A -85,B 0,C 180,E1 -7070.647,E2 -7070.647} C_VEL
LIN {X 0,Y 481.581,Z 214.499,A -85,B 0,C 180,E1 -7073.371,E2 -7073.371} C_VEL
LIN {X 0,Y 481.654,Z 214.483,A -85,B 0,C 180,E1 -7076.327,E2 -7076.327} C_VEL
LIN {X 0,Y 481.6,Z 214.495,A -85,B 0,C 180,E1 -7079.413,E2 -7079.413} C_VEL
LIN {X 0,Y 481.643,Z 214.484,A -85,B 0,C 180,E1 -7082.165,E2 -7082.165} C_VEL
LIN {X 0,Y 481.661,Z 214.488,A -85,B 0,C 180,E1 -7084.967,E2 -7084.967} C_VEL
LIN {X 0,Y 481.603,Z 214.49,A -85,B 0,C 180,E1 -7087.931,E2 -7087.931} C_VEL
LIN {X 0,Y 480.932,Z 214.576,A -85,B 0,C 180,E1 -7088.629,E2 -7088.629} C_VEL
LIN {X 0,Y 478.096,Z 214.931,A -85,B 0,C 180,E1 -7089.763,E2 -7089.763} C_VEL
LIN {X 0,Y 475.705,Z 215.231,A -85,B 0,C 180,E1 -7090.678,E2 -7090.678} C_VEL
LIN {X 0,Y 474.684,Z 215.357,A -85,B 0,C 180,E1 -7091.383,E2 -7091.383} C_VEL
LIN {X 0,Y 474.603,Z 215.364,A -85,B 0,C 180,E1 -7091.622,E2 -7091.622} C_VEL
LIN {X 0,Y 474.636,Z 215.359,A -85,B 0,C 180,E1 -7094.543,E2 -7094.543} C_VEL
LIN {X 0,Y 474.675,Z 215.352,A -85,B 0,C 180,E1 -7098.037,E2 -7098.037} C_VEL
LIN {X 0,Y 474.683,Z 215.355,A -85,B 0,C 180,E1 -7101.486,E2 -7101.486} C_VEL
LIN {X 0,Y 474.735,Z 215.345,A -85,B 0,C 180,E1 -7104.052,E2 -7104.052} C_VEL
LIN {X 0,Y 474.836,Z 215.336,A -85,B 0,C 180,E1 -7107.455,E2 -7107.455} C_VEL
LIN {X 0,Y 474.843,Z 215.332,A -85,B 0,C 180,E1 -7110,E2 -7110} C_VEL
LIN {X 0,Y 474.836,Z 215.335,A -85,B 0,C 180,E1 -7112.545,E2 -7112.545} C_VEL
LIN {X 0,Y 474.735,Z 215.345,A -85,B 0,C 180,E1 -7115.948,E2 -7115.948} C_VEL
LIN {X 0,Y 474.683,Z 215.355,A -85,B 0,C 180,E1 -7118.514,E2 -7118.514} C_VEL
LIN {X 0,Y 474.705,Z 215.426,A -85,B 0,C 180,E1 -7122.264,E2 -7122.264} C_VEL
LIN {X 0,Y 475.69,Z 223.041,A -85,B 0,C 180,E1 -7123.891,E2 -7123.891} C_VEL
LIN {X 0,Y 475.376,Z 234.933,A -85,B 0,C 180,E1 -7126.313,E2 -7126.313} C_VEL
LIN {X 0,Y 478.167,Z 249.951,A -85,B 0,C 180,E1 -7126.654,E2 -7126.654} C_VEL
LIN {X 0,Y 477.367,Z 342.483,A -85,B 0,C 180,E1 -7128.092,E2 -7128.092} C_VEL
LIN {X 0,Y 477.074,Z 356.278,A -85,B 0,C 180,E1 -7128.492,E2 -7128.492} C_VEL
LIN {X 0,Y 476.761,Z 368.829,A -85,B 0,C 180,E1 -7129.037,E2 -7129.037} C_VEL
LIN {X 0,Y 476.339,Z 381.056,A -85,B 0,C 180,E1 -7129.76,E2 -7129.76} C_VEL
LIN {X 0,Y 475.892,Z 392.675,A -85,B 0,C 180,E1 -7130.645,E2 -7130.645} C_VEL
LIN {X 0,Y 475.443,Z 401.578,A -85,B 0,C 180,E1 -7131.484,E2 -7131.484} C_VEL
LIN {X 0,Y 474.982,Z 411.429,A -85,B 0,C 180,E1 -7132.625,E2 -7132.625} C_VEL
LIN {X 0,Y 474.643,Z 419.62,A -85,B 0,C 180,E1 -7133.796,E2 -7133.796} C_VEL
LIN {X 0,Y 474.355,Z 427.2,A -85,B 0,C 180,E1 -7135.134,E2 -7135.134} C_VEL
LIN {X 0,Y 474.08,Z 432.939,A -85,B 0,C 180,E1 -7136.406,E2 -7136.406} C_VEL
LIN {X 0,Y 473.905,Z 437.968,A -85,B 0,C 180,E1 -7137.848,E2 -7137.848} C_VEL
LIN {X 0,Y 473.793,Z 441.681,A -85,B 0,C 180,E1 -7139.307,E2 -7139.307} C_VEL
LIN {X 0,Y 473.671,Z 443.963,A -85,B 0,C 180,E1 -7140.635,E2 -7140.635} C_VEL
LIN {X 0,Y 473.612,Z 445.435,A -85,B 0,C 180,E1 -7142.289,E2 -7142.289} C_VEL
LIN {X 0,Y 473.616,Z 445.444,A -85,B 0,C 180,E1 -7143.814,E2 -7143.814} C_VEL
LIN {X 0,Y 473.651,Z 444.14,A -85,B 0,C 180,E1 -7145.357,E2 -7145.357} C_VEL
LIN {X 0,Y 473.766,Z 441.76,A -85,B 0,C 180,E1 -7146.782,E2 -7146.782} C_VEL
LIN {X 0,Y 473.932,Z 438.186,A -85,B 0,C 180,E1 -7148.204,E2 -7148.204} C_VEL
LIN {X 0,Y 474.085,Z 433.409,A -85,B 0,C 180,E1 -7149.6,E2 -7149.6} C_VEL
LIN {X 0,Y 474.353,Z 426.665,A -85,B 0,C 180,E1 -7151.094,E2 -7151.094} C_VEL
LIN {X 0,Y 474.639,Z 420.125,A -85,B 0,C 180,E1 -7152.25,E2 -7152.25} C_VEL
LIN {X 0,Y 475.111,Z 410.989,A -85,B 0,C 180,E1 -7153.556,E2 -7153.556} C_VEL
LIN {X 0,Y 475.507,Z 402.044,A -85,B 0,C 180,E1 -7154.59,E2 -7154.59} C_VEL
LIN {X 0,Y 475.94,Z 391.366,A -85,B 0,C 180,E1 -7155.587,E2 -7155.587} C_VEL
LIN {X 0,Y 476.459,Z 379.94,A -85,B 0,C 180,E1 -7156.435,E2 -7156.435} C_VEL
LIN {X 0,Y 476.85,Z 368.874,A -85,B 0,C 180,E1 -7157.079,E2 -7157.079} C_VEL
LIN {X 0,Y 477.184,Z 356.223,A -85,B 0,C 180,E1 -7157.624,E2 -7157.624} C_VEL
LIN {X 0,Y 477.415,Z 342.554,A -85,B 0,C 180,E1 -7158.021,E2 -7158.021} C_VEL
LIN {X 0,Y 478.17,Z 248.656,A -85,B 0,C 180,E1 -7159.488,E2 -7159.488} C_VEL
LIN {X 0,Y 475.438,Z 234.847,A -85,B 0,C 180,E1 -7159.826,E2 -7159.826} C_VEL
LIN {X 0,Y 475.59,Z 221.032,A -85,B 0,C 180,E1 -7162.45,E2 -7162.45} C_VEL
LIN {X 0,Y 474.635,Z 215.365,A -85,B 0,C 180,E1 -7163.596,E2 -7163.596} C_VEL
LIN {X 0,Y 474.604,Z 215.369,A -85,B 0,C 180,E1 -7166.785,E2 -7166.785} C_VEL
LIN {X 0,Y 474.577,Z 215.369,A -85,B 0,C 180,E1 -7169.775,E2 -7169.775} C_VEL
LIN {X 0,Y 474.681,Z 215.357,A -85,B 0,C 180,E1 -7172.686,E2 -7172.686} C_VEL
LIN {X 0,Y 474.627,Z 215.362,A -85,B 0,C 180,E1 -7175.512,E2 -7175.512} C_VEL
LIN {X 0,Y 474.642,Z 215.364,A -85,B 0,C 180,E1 -7179.191,E2 -7179.191} C_VEL
LIN {X 0,Y 474.631,Z 215.361,A -85,B 0,C 180,E1 -7181.889,E2 -7181.889} C_VEL
LIN {X 0,Y 474.676,Z 215.359,A -85,B 0,C 180,E1 -7184.549,E2 -7184.549} C_VEL
LIN {X 0,Y 474.719,Z 215.348,A -85,B 0,C 180,E1 -7188.044,E2 -7188.044} C_VEL
LIN {X 0,Y 474.694,Z 215.35,A -85,B 0,C 180,E1 -7191.491,E2 -7191.491} C_VEL
LIN {X 0,Y 474.749,Z 215.344,A -85,B 0,C 180,E1 -7194.057,E2 -7194.057} C_VEL
LIN {X 0,Y 474.876,Z 215.328,A -85,B 0,C 180,E1 -7197.46,E2 -7197.46} C_VEL
LIN {X 0,Y 474.894,Z 215.326,A -85,B 0,C 180,E1 -7200.005,E2 -7200.005} C_VEL
LIN {X 0,Y 474.868,Z 215.331,A -85,B 0,C 180,E1 -7202.549,E2 -7202.549} C_VEL
LIN {X 0,Y 474.749,Z 215.341,A -85,B 0,C 180,E1 -7205.952,E2 -7205.952} C_VEL
LIN {X 0,Y 474.694,Z 215.357,A -85,B 0,C 180,E1 -7208.518,E2 -7208.518} C_VEL
LIN {X 0,Y 474.698,Z 215.351,A -85,B 0,C 180,E1 -7211.967,E2 -7211.967} C_VEL
LIN {X 0,Y 474.695,Z 215.351,A -85,B 0,C 180,E1 -7215.46,E2 -7215.46} C_VEL
LIN {X 0,Y 474.659,Z 215.357,A -85,B 0,C 180,E1 -7219.014,E2 -7219.014} C_VEL
LIN {X 0,Y 474.587,Z 215.363,A -85,B 0,C 180,E1 -7221.733,E2 -7221.733} C_VEL
LIN {X 0,Y 474.62,Z 215.367,A -85,B 0,C 180,E1 -7224.499,E2 -7224.499} C_VEL
LIN {X 0,Y 474.595,Z 215.363,A -85,B 0,C 180,E1 -7227.33,E2 -7227.33} C_VEL
LIN {X 0,Y 474.597,Z 215.366,A -85,B 0,C 180,E1 -7230.234,E2 -7230.234} C_VEL
LIN {X 0,Y 474.617,Z 215.358,A -85,B 0,C 180,E1 -7233.226,E2 -7233.226} C_VEL
LIN {X 0,Y 474.572,Z 215.372,A -85,B 0,C 180,E1 -7236.328,E2 -7236.328} C_VEL
LIN {X 0,Y 474.603,Z 215.362,A -85,B 0,C 180,E1 -7239.553,E2 -7239.553} C_VEL
LIN {X 0,Y 474.57,Z 215.37,A -85,B 0,C 180,E1 -7242.943,E2 -7242.943} C_VEL
LIN {X 0,Y 474.572,Z 215.371,A -85,B 0,C 180,E1 -7245.892,E2 -7245.892} C_VEL
LIN {X 0,Y 474.585,Z 215.366,A -85,B 0,C 180,E1 -7249.05,E2 -7249.05} C_VEL
LIN {X 0,Y 474.588,Z 215.367,A -85,B 0,C 180,E1 -7251.711,E2 -7251.711} C_VEL
LIN {X 0,Y 474.606,Z 215.366,A -85,B 0,C 180,E1 -7254.725,E2 -7254.725} C_VEL
LIN {X 0,Y 474.616,Z 215.367,A -85,B 0,C 180,E1 -7257.787,E2 -7257.787} C_VEL
LIN {X 0,Y 474.58,Z 215.371,A -85,B 0,C 180,E1 -7260.898,E2 -7260.898} C_VEL
LIN {X 0,Y 474.585,Z 215.372,A -85,B 0,C 180,E1 -7264.098,E2 -7264.098} C_VEL
LIN {X 0,Y 474.612,Z 215.51,A -85,B 0,C 180,E1 -7264.326,E2 -7264.326} C_VEL
LIN {X 0,Y 476.634,Z 226.093,A -85,B 0,C 180,E1 -7266.269,E2 -7266.269} C_VEL
LIN {X 0,Y 476.158,Z 241.017,A -85,B 0,C 180,E1 -7268.81,E2 -7268.81} C_VEL
LIN {X 0,Y 475.516,Z 259.528,A -85,B 0,C 180,E1 -7271.919,E2 -7271.919} C_VEL
LIN {X 0,Y 475.248,Z 267.34,A -85,B 0,C 180,E1 -7273.219,E2 -7273.219} C_VEL
LIN {X 0,Y 477.984,Z 285.964,A -85,B 0,C 180,E1 -7273.612,E2 -7273.612} C_VEL
LIN {X 0,Y 477.365,Z 376.002,A -85,B 0,C 180,E1 -7275.016,E2 -7275.016} C_VEL
LIN {X 0,Y 476.972,Z 389.206,A -85,B 0,C 180,E1 -7275.385,E2 -7275.385} C_VEL
LIN {X 0,Y 476.559,Z 401.926,A -85,B 0,C 180,E1 -7275.917,E2 -7275.917} C_VEL
LIN {X 0,Y 476.088,Z 413.251,A -85,B 0,C 180,E1 -7276.556,E2 -7276.556} C_VEL
LIN {X 0,Y 475.66,Z 424.402,A -85,B 0,C 180,E1 -7277.367,E2 -7277.367} C_VEL
LIN {X 0,Y 475.182,Z 435.483,A -85,B 0,C 180,E1 -7278.375,E2 -7278.375} C_VEL
LIN {X 0,Y 474.746,Z 444.096,A -85,B 0,C 180,E1 -7279.337,E2 -7279.337} C_VEL
LIN {X 0,Y 474.428,Z 452.049,A -85,B 0,C 180,E1 -7280.407,E2 -7280.407} C_VEL
LIN {X 0,Y 474.141,Z 459.822,A -85,B 0,C 180,E1 -7281.691,E2 -7281.691} C_VEL
LIN {X 0,Y 473.905,Z 466.98,A -85,B 0,C 180,E1 -7283.187,E2 -7283.187} C_VEL
LIN {X 0,Y 473.841,Z 471.749,A -85,B 0,C 180,E1 -7284.468,E2 -7284.468} C_VEL
LIN {X 0,Y 473.737,Z 475.393,A -85,B 0,C 180,E1 -7285.746,E2 -7285.746} C_VEL
LIN {X 0,Y 473.799,Z 477.278,A -85,B 0,C 180,E1 -7286.599,E2 -7286.599} C_VEL
LIN {X 0,Y 473.745,Z 478.689,A -85,B 0,C 180,E1 -7287.449,E2 -7287.449} C_VEL
LIN {X 0,Y 473.728,Z 479.698,A -85,B 0,C 180,E1 -7288.3,E2 -7288.3} C_VEL
LIN {X 0,Y 473.693,Z 480.316,A -85,B 0,C 180,E1 -7289.15,E2 -7289.15} C_VEL
LIN {X 0,Y 473.677,Z 480.538,A -85,B 0,C 180,E1 -7290,E2 -7290} C_VEL
LIN {X 0,Y 473.693,Z 480.325,A -85,B 0,C 180,E1 -7290.85,E2 -7290.85} C_VEL
LIN {X 0,Y 473.728,Z 479.719,A -85,B 0,C 180,E1 -7291.7,E2 -7291.7} C_VEL
LIN {X 0,Y 473.745,Z 478.721,A -85,B 0,C 180,E1 -7292.551,E2 -7292.551} C_VEL
LIN {X 0,Y 473.799,Z 477.318,A -85,B 0,C 180,E1 -7293.402,E2 -7293.402} C_VEL
LIN {X 0,Y 473.763,Z 474.364,A -85,B 0,C 180,E1 -7294.68,E2 -7294.68} C_VEL
LIN {X 0,Y 473.828,Z 470.364,A -85,B 0,C 180,E1 -7295.959,E2 -7295.959} C_VEL
LIN {X 0,Y 474.012,Z 464.206,A -85,B 0,C 180,E1 -7297.454,E2 -7297.454} C_VEL
LIN {X 0,Y 474.256,Z 457.481,A -85,B 0,C 180,E1 -7298.737,E2 -7298.737} C_VEL
LIN {X 0,Y 474.548,Z 449.135,A -85,B 0,C 180,E1 -7300.021,E2 -7300.021} C_VEL
LIN {X 0,Y 474.965,Z 440.559,A -85,B 0,C 180,E1 -7301.09,E2 -7301.09} C_VEL
LIN {X 0,Y 475.445,Z 430.262,A -85,B 0,C 180,E1 -7302.133,E2 -7302.133} C_VEL
LIN {X 0,Y 475.815,Z 419.772,A -85,B 0,C 180,E1 -7302.995,E2 -7302.995} C_VEL
LIN {X 0,Y 476.29,Z 407.947,A -85,B 0,C 180,E1 -7303.764,E2 -7303.764} C_VEL
LIN {X 0,Y 476.742,Z 395.991,A -85,B 0,C 180,E1 -7304.35,E2 -7304.35} C_VEL
LIN {X 0,Y 477.103,Z 383.09,A -85,B 0,C 180,E1 -7304.802,E2 -7304.802} C_VEL
LIN {X 0,Y 477.403,Z 369.499,A -85,B 0,C 180,E1 -7305.092,E2 -7305.092} C_VEL
LIN {X 0,Y 477.865,Z 284.796,A -85,B 0,C 180,E1 -7306.394,E2 -7306.394} C_VEL
LIN {X 0,Y 475.272,Z 267.796,A -85,B 0,C 180,E1 -7306.759,E2 -7306.759} C_VEL
LIN {X 0,Y 475.886,Z 250.99,A -85,B 0,C 180,E1 -7309.609,E2 -7309.609} C_VEL
LIN {X 0,Y 476.62,Z 233.891,A -85,B 0,C 180,E1 -7312.543,E2 -7312.543} C_VEL
LIN {X 0,Y 476.793,Z 226.754,A -85,B 0,C 180,E1 -7313.788,E2 -7313.788} C_VEL
LIN {X 0,Y 474.603,Z 215.369,A -85,B 0,C 180,E1 -7315.96,E2 -7315.96} C_VEL
LIN {X 0,Y 474.576,Z 215.37,A -85,B 0,C 180,E1 -7319.254,E2 -7319.254} C_VEL
LIN {X 0,Y 474.581,Z 215.365,A -85,B 0,C 180,E1 -7322.42,E2 -7322.42} C_VEL
LIN {X 0,Y 474.564,Z 215.37,A -85,B 0,C 180,E1 -7325.457,E2 -7325.457} C_VEL
LIN {X 0,Y 474.585,Z 215.365,A -85,B 0,C 180,E1 -7328.459,E2 -7328.459} C_VEL
LIN {X 0,Y 474.581,Z 215.373,A -85,B 0,C 180,E1 -7331.788,E2 -7331.788} C_VEL
LIN {X 0,Y 474.59,Z 215.366,A -85,B 0,C 180,E1 -7335.299,E2 -7335.299} C_VEL
LIN {X 0,Y 474.584,Z 215.366,A -85,B 0,C 180,E1 -7338.207,E2 -7338.207} C_VEL
LIN {X 0,Y 474.581,Z 215.37,A -85,B 0,C 180,E1 -7341.536,E2 -7341.536} C_VEL
LIN {X 0,Y 474.568,Z 215.366,A -85,B 0,C 180,E1 -7344.717,E2 -7344.717} C_VEL
LIN {X 0,Y 474.611,Z 215.368,A -85,B 0,C 180,E1 -7347.782,E2 -7347.782} C_VEL
LIN {X 0,Y 474.573,Z 215.366,A -85,B 0,C 180,E1 -7350.893,E2 -7350.893} C_VEL
LIN {X 0,Y 474.556,Z 215.376,A -85,B 0,C 180,E1 -7353.619,E2 -7353.619} C_VEL
LIN {X 0,Y 474.634,Z 215.358,A -85,B 0,C 180,E1 -7356.639,E2 -7356.639} C_VEL
LIN {X 0,Y 474.612,Z 215.363,A -85,B 0,C 180,E1 -7360.084,E2 -7360.084} C_VEL
LIN {X 0,Y 474.606,Z 215.361,A -85,B 0,C 180,E1 -7362.769,E2 -7362.769} C_VEL
LIN {X 0,Y 474.628,Z 215.364,A -85,B 0,C 180,E1 -7365.416,E2 -7365.416} C_VEL
LIN {X 0,Y 474.67,Z 215.356,A -85,B 0,C 180,E1 -7368.033,E2 -7368.033} C_VEL
LIN {X 0,Y 474.652,Z 215.363,A -85,B 0,C 180,E1 -7371.481,E2 -7371.481} C_VEL
LIN {X 0,Y 474.727,Z 215.348,A -85,B 0,C 180,E1 -7374.047,E2 -7374.047} C_VEL
LIN {X 0,Y 474.832,Z 215.34,A -85,B 0,C 180,E1 -7377.45,E2 -7377.45} C_VEL
LIN {X 0,Y 474.863,Z 215.331,A -85,B 0,C 180,E1 -7379.995,E2 -7379.995} C_VEL
LIN {X 0,Y 474.864,Z 215.329,A -85,B 0,C 180,E1 -7382.54,E2 -7382.54} C_VEL
LIN {X 0,Y 474.71,Z 215.351,A -85,B 0,C 180,E1 -7385.943,E2 -7385.943} C_VEL
LIN {X 0,Y 474.648,Z 215.356,A -85,B 0,C 180,E1 -7388.51,E2 -7388.51} C_VEL
LIN {X 0,Y 474.682,Z 215.354,A -85,B 0,C 180,E1 -7391.957,E2 -7391.957} C_VEL
LIN {X 0,Y 474.655,Z 215.359,A -85,B 0,C 180,E1 -7395.762,E2 -7395.762} C_VEL
LIN {X 0,Y 474.634,Z 215.361,A -85,B 0,C 180,E1 -7399.005,E2 -7399.005} C_VEL
LIN {X 0,Y 474.558,Z 215.371,A -85,B 0,C 180,E1 -7401.724,E2 -7401.724} C_VEL
LIN {X 0,Y 474.595,Z 215.362,A -85,B 0,C 180,E1 -7404.49,E2 -7404.49} C_VEL
LIN {X 0,Y 474.64,Z 215.365,A -85,B 0,C 180,E1 -7407.327,E2 -7407.327} C_VEL
LIN {X 0,Y 474.566,Z 215.366,A -85,B 0,C 180,E1 -7410.225,E2 -7410.225} C_VEL
LIN {X 0,Y 474.595,Z 215.369,A -85,B 0,C 180,E1 -7413.216,E2 -7413.216} C_VEL
LIN {X 0,Y 474.546,Z 215.368,A -85,B 0,C 180,E1 -7416.319,E2 -7416.319} C_VEL
LIN {X 0,Y 474.583,Z 215.368,A -85,B 0,C 180,E1 -7419.643,E2 -7419.643} C_VEL
LIN {X 0,Y 474.568,Z 215.369,A -85,B 0,C 180,E1 -7422.93,E2 -7422.93} C_VEL
LIN {X 0,Y 474.56,Z 215.368,A -85,B 0,C 180,E1 -7425.891,E2 -7425.891} C_VEL
LIN {X 0,Y 474.577,Z 215.37,A -85,B 0,C 180,E1 -7429.037,E2 -7429.037} C_VEL
LIN {X 0,Y 474.558,Z 215.37,A -85,B 0,C 180,E1 -7431.7,E2 -7431.7} C_VEL
LIN {X 0,Y 474.577,Z 215.367,A -85,B 0,C 180,E1 -7434.723,E2 -7434.723} C_VEL
LIN {X 0,Y 474.579,Z 215.366,A -85,B 0,C 180,E1 -7437.784,E2 -7437.784} C_VEL
LIN {X 0,Y 474.573,Z 215.369,A -85,B 0,C 180,E1 -7440.88,E2 -7440.88} C_VEL
LIN {X 0,Y 474.607,Z 215.364,A -85,B 0,C 180,E1 -7443.626,E2 -7443.626} C_VEL
LIN {X 0,Y 474.592,Z 215.365,A -85,B 0,C 180,E1 -7446.634,E2 -7446.634} C_VEL
LIN {X 0,Y 474.614,Z 215.368,A -85,B 0,C 180,E1 -7449.183,E2 -7449.183} C_VEL
LIN {X 0,Y 474.603,Z 215.364,A -85,B 0,C 180,E1 -7451.622,E2 -7451.622} C_VEL
LIN {X 0,Y 473.943,Z 215.445,A -85,B 0,C 180,E1 -7452.331,E2 -7452.331} C_VEL
LIN {X 0,Y 471.089,Z 215.806,A -85,B 0,C 180,E1 -7453.483,E2 -7453.483} C_VEL
LIN {X 0,Y 468.668,Z 216.111,A -85,B 0,C 180,E1 -7454.411,E2 -7454.411} C_VEL
LIN {X 0,Y 467.624,Z 216.239,A -85,B 0,C 180,E1 -7455.128,E2 -7455.128} C_VEL
LIN {X 0,Y 467.536,Z 216.247,A -85,B 0,C 180,E1 -7455.371,E2 -7455.371} C_VEL
LIN {X 0,Y 467.634,Z 216.23,A -85,B 0,C 180,E1 -7457.854,E2 -7457.854} C_VEL
LIN {X 0,Y 467.632,Z 216.234,A -85,B 0,C 180,E1 -7461.357,E2 -7461.357} C_VEL
